(* CODESYS project T620X_PLC_CR711S.project
   Title: T620X PLC
   Description: T620X PLC - pwm ramp mods / sim mods - link fixed for RAMP_LIMIT to the output block
   Version: 1.0.3.0
   Company: Mtech

Project tree, tasks and I/O mapping:
  SafetyPLC : CR711S SIL2, ifm electronic, order no. CR711S, version 3.2.0.0
    application Application
      libraries: ifmR360-3, * (ifm electronic); Standard, * (System); Util, * (System)
      task Task (cyclic, interval t#10ms, priority 1, watchdog t#8ms x 1) calls PLC_PRG
      global variables EVL
      program PLC_PRG [FBD]
    Communication : Communication, ifm electronic, version 3.2.0.0
      CAN : CAN, ifm electronic, version 3.2.0.0
      Ethernet : Ethernet, ifm electronic, version 3.2.0.0
    HMI : HMI, ifm electronic, version 3.2.0.0
      User_LEDs : User_LEDs, ifm electronic, version 3.2.0.0
          input  UserLED0_I : LED_IEC_B_INPUT_MAPPING_TYPE  // UserLED0_I
          input  UserLED1_I : LED_IEC_B_INPUT_MAPPING_TYPE  // UserLED1_I
          input  UserLED2_I : LED_IEC_B_INPUT_MAPPING_TYPE  // UserLED2_I
          input  UserLED3_I : LED_IEC_B_INPUT_MAPPING_TYPE  // UserLED3_I
          output UserLED0_Q : LED_IEC_B_OUTPUT_MAPPING_TYPE  // User LED 0
          output UserLED1_Q : LED_IEC_B_OUTPUT_MAPPING_TYPE  // User LED 1
          output UserLED2_Q : LED_IEC_B_OUTPUT_MAPPING_TYPE  // User LED 2
          output UserLED3_Q : LED_IEC_B_OUTPUT_MAPPING_TYPE  // User LED 3
    Local_IO : Local_IO, ifm electronic, version 3.2.0.0
      Inputs : Inputs, ifm electronic, version 3.2.0.0
          input  IN0100_I : IN_MULTIFUNCTION_A_INPUT_MAPPING_TYPE  // IN0100_I
          input  IN0101_I : IN_MULTIFUNCTION_A_INPUT_MAPPING_TYPE  // IN0101_I
          input  IN0102_I : IN_MULTIFUNCTION_A_INPUT_MAPPING_TYPE  // IN0102_I
          input  IN0103_I : IN_MULTIFUNCTION_A_INPUT_MAPPING_TYPE  // IN0103_I
          input  IN0200_I : IN_MULTIFUNCTION_A_INPUT_MAPPING_TYPE  // IN0200_I
          input  IN0201_I : IN_MULTIFUNCTION_A_INPUT_MAPPING_TYPE  // IN0201_I
          input  IN0202_I : IN_MULTIFUNCTION_A_INPUT_MAPPING_TYPE  // IN0202_I
          input  IN0203_I : IN_MULTIFUNCTION_A_INPUT_MAPPING_TYPE  // IN0203_I
          input  IN0600_I : IN_MULTIFUNCTION_A_INPUT_MAPPING_TYPE  // IN0600_I
          input  IN0601_I : IN_MULTIFUNCTION_A_INPUT_MAPPING_TYPE  // IN0601_I
          input  IN0602_I : IN_MULTIFUNCTION_A_INPUT_MAPPING_TYPE  // IN0602_I
          input  IN0603_I : IN_MULTIFUNCTION_A_INPUT_MAPPING_TYPE  // IN0603_I
          input  IN0700_I : IN_MULTIFUNCTION_A_INPUT_MAPPING_TYPE  // IN0700_I
          input  IN0701_I : IN_MULTIFUNCTION_A_INPUT_MAPPING_TYPE  // IN0701_I
          input  IN0702_I : IN_MULTIFUNCTION_A_INPUT_MAPPING_TYPE  // IN0702_I
          input  IN0703_I : IN_MULTIFUNCTION_A_INPUT_MAPPING_TYPE  // IN0703_I
          input  IN0400_I : IN_RESISTOR_A_INPUT_MAPPING_TYPE  // IN0400_I
          input  IN0401_I : IN_RESISTOR_A_INPUT_MAPPING_TYPE  // IN0401_I
          input  IN0900_I : IN_RESISTOR_A_INPUT_MAPPING_TYPE  // IN0900_I
          input  IN0901_I : IN_RESISTOR_A_INPUT_MAPPING_TYPE  // IN0901_I
          input  IN0300_I : IN_DIGITAL_B_INPUT_MAPPING_TYPE  // IN0300_I
          input  IN0301_I : IN_DIGITAL_B_INPUT_MAPPING_TYPE  // IN0301_I
          input  IN0800_I : IN_DIGITAL_B_INPUT_MAPPING_TYPE  // IN0800_I
          input  IN0801_I : IN_DIGITAL_B_INPUT_MAPPING_TYPE  // IN0801_I
          input  COM_RESET_I : IN_COMMUNICATION_RESET_INPUT_MAPPING_TYPE  // COM_RESET_I
          input  IN0000_I : IN_FREQUENCY_B_CHANNEL_A_INPUT_MAPPING_TYPE  // IN0000_I
          input  IN0002_I : IN_FREQUENCY_B_CHANNEL_A_INPUT_MAPPING_TYPE  // IN0002_I
          input  IN0500_I : IN_FREQUENCY_B_CHANNEL_A_INPUT_MAPPING_TYPE  // IN0500_I
          input  IN0502_I : IN_FREQUENCY_B_CHANNEL_A_INPUT_MAPPING_TYPE  // IN0502_I
          input  IN0001_I : IN_FREQUENCY_B_CHANNEL_B_INPUT_MAPPING_TYPE  // IN0001_I
          input  IN0003_I : IN_FREQUENCY_B_CHANNEL_B_INPUT_MAPPING_TYPE  // IN0003_I
          input  IN0501_I : IN_FREQUENCY_B_CHANNEL_B_INPUT_MAPPING_TYPE  // IN0501_I
          input  IN0503_I : IN_FREQUENCY_B_CHANNEL_B_INPUT_MAPPING_TYPE  // IN0503_I
      Outputs : Outputs, ifm electronic, version 3.2.0.0
          input  OUT0006_I : OUT_PWM_40_BRIDGE_A_INPUT_MAPPING_TYPE  // OUT0006_I
          input  OUT0106_I : OUT_PWM_40_BRIDGE_A_INPUT_MAPPING_TYPE  // OUT0106_I
          input  OUT0206_I : OUT_PWM_40_BRIDGE_A_INPUT_MAPPING_TYPE  // OUT0206_I
          input  OUT0008_I : OUT_PWM_40_A_INPUT_MAPPING_TYPE  // OUT0008_I
          input  OUT0108_I : OUT_PWM_40_A_INPUT_MAPPING_TYPE  // OUT0108_I
          input  OUT0208_I : OUT_PWM_40_A_INPUT_MAPPING_TYPE  // OUT0208_I
          input  OUT0000_I : OUT_PWM_25_A_INPUT_MAPPING_TYPE  // OUT0000_I
          input  OUT0002_I : OUT_PWM_25_A_INPUT_MAPPING_TYPE  // OUT0002_I
          input  OUT0004_I : OUT_PWM_25_A_INPUT_MAPPING_TYPE  // OUT0004_I
          input  OUT0100_I : OUT_PWM_25_A_INPUT_MAPPING_TYPE  // OUT0100_I
          input  OUT0102_I : OUT_PWM_25_A_INPUT_MAPPING_TYPE  // OUT0102_I
          input  OUT0104_I : OUT_PWM_25_A_INPUT_MAPPING_TYPE  // OUT0104_I
          input  OUT0200_I : OUT_PWM_25_A_INPUT_MAPPING_TYPE  // OUT0200_I
          input  OUT0202_I : OUT_PWM_25_A_INPUT_MAPPING_TYPE  // OUT0202_I
          input  OUT0204_I : OUT_PWM_25_A_INPUT_MAPPING_TYPE  // OUT0204_I
          input  OUT3001_I : OUT_VOLTAGE_A_INPUT_MAPPING_TYPE  // OUT3001_I
          input  OUT3000_I : OUT_SUPPLY_A_INPUT_MAPPING_TYPE  // OUT3000_I
          input  OUT0001_I : OUT_PWM_25_B_INPUT_MAPPING_TYPE  // OUT0001_I
          input  OUT0003_I : OUT_PWM_25_B_INPUT_MAPPING_TYPE  // OUT0003_I
          input  OUT0005_I : OUT_PWM_25_B_INPUT_MAPPING_TYPE  // OUT0005_I
          input  OUT0101_I : OUT_PWM_25_B_INPUT_MAPPING_TYPE  // OUT0101_I
          input  OUT0103_I : OUT_PWM_25_B_INPUT_MAPPING_TYPE  // OUT0103_I
          input  OUT0105_I : OUT_PWM_25_B_INPUT_MAPPING_TYPE  // OUT0105_I
          input  OUT0201_I : OUT_PWM_25_B_INPUT_MAPPING_TYPE  // OUT0201_I
          input  OUT0203_I : OUT_PWM_25_B_INPUT_MAPPING_TYPE  // OUT0203_I
          input  OUT0205_I : OUT_PWM_25_B_INPUT_MAPPING_TYPE  // OUT0205_I
          input  OUT0007_I : OUT_PWM_40_BRIDGE_A_INPUT_MAPPING_TYPE  // OUT0007_I
          input  OUT0107_I : OUT_PWM_40_BRIDGE_A_INPUT_MAPPING_TYPE  // OUT0107_I
          input  OUT0207_I : OUT_PWM_40_BRIDGE_A_INPUT_MAPPING_TYPE  // OUT0207_I
          output OUT0006_Q : OUT_PWM_40_BRIDGE_A_OUTPUT_MAPPING_TYPE  // OUT0006_Q
          output OUT0106_Q : OUT_PWM_40_BRIDGE_A_OUTPUT_MAPPING_TYPE  // OUT0106_Q
          output OUT0206_Q : OUT_PWM_40_BRIDGE_A_OUTPUT_MAPPING_TYPE  // OUT0206_Q
          output OUT0008_Q : OUT_PWM_40_A_OUTPUT_MAPPING_TYPE  // OUT0008_Q
          output OUT0108_Q : OUT_PWM_40_A_OUTPUT_MAPPING_TYPE  // OUT0108_Q
          output OUT0208_Q : OUT_PWM_40_A_OUTPUT_MAPPING_TYPE  // OUT0208_Q
          output OUT0000_Q : OUT_PWM_25_A_OUTPUT_MAPPING_TYPE  // OUT0000_Q
          output OUT0002_Q : OUT_PWM_25_A_OUTPUT_MAPPING_TYPE  // OUT0002_Q
          output OUT0004_Q : OUT_PWM_25_A_OUTPUT_MAPPING_TYPE  // OUT0004_Q
          output OUT0100_Q : OUT_PWM_25_A_OUTPUT_MAPPING_TYPE  // OUT0100_Q
          output OUT0102_Q : OUT_PWM_25_A_OUTPUT_MAPPING_TYPE  // OUT0102_Q
          output OUT0104_Q : OUT_PWM_25_A_OUTPUT_MAPPING_TYPE  // OUT0104_Q
          output OUT0200_Q : OUT_PWM_25_A_OUTPUT_MAPPING_TYPE  // OUT0200_Q
          output OUT0202_Q : OUT_PWM_25_A_OUTPUT_MAPPING_TYPE  // OUT0202_Q
          output OUT0204_Q : OUT_PWM_25_A_OUTPUT_MAPPING_TYPE  // OUT0204_Q
          output OUT3001_Q : OUT_VOLTAGE_A_OUTPUT_MAPPING_TYPE  // OUT3001_Q
          output OUT3000_Q : OUT_SUPPLY_A_OUTPUT_MAPPING_TYPE  // OUT3000_Q
          output OUT0001_Q : OUT_PWM_25_B_OUTPUT_MAPPING_TYPE  // OUT0001_Q
          output OUT0003_Q : OUT_PWM_25_B_OUTPUT_MAPPING_TYPE  // OUT0003_Q
          output OUT0005_Q : OUT_PWM_25_B_OUTPUT_MAPPING_TYPE  // OUT0005_Q
          output OUT0101_Q : OUT_PWM_25_B_OUTPUT_MAPPING_TYPE  // OUT0101_Q
          output OUT0103_Q : OUT_PWM_25_B_OUTPUT_MAPPING_TYPE  // OUT0103_Q
          output OUT0105_Q : OUT_PWM_25_B_OUTPUT_MAPPING_TYPE  // OUT0105_Q
          output OUT0201_Q : OUT_PWM_25_B_OUTPUT_MAPPING_TYPE  // OUT0201_Q
          output OUT0203_Q : OUT_PWM_25_B_OUTPUT_MAPPING_TYPE  // OUT0203_Q
          output OUT0205_Q : OUT_PWM_25_B_OUTPUT_MAPPING_TYPE  // OUT0205_Q
          output OUT0007_Q : OUT_PWM_40_BRIDGE_A_OUTPUT_MAPPING_TYPE  // OUT0007_Q
          output OUT0107_Q : OUT_PWM_40_BRIDGE_A_OUTPUT_MAPPING_TYPE  // OUT0107_Q
          output OUT0207_Q : OUT_PWM_40_BRIDGE_A_OUTPUT_MAPPING_TYPE  // OUT0207_Q
      System_Inputs : System_Inputs, ifm electronic, version 3.2.0.0
          input  VBB30 : IN_SYSTEM_VOLTAGE_INPUT_MAPPING_TYPE  // VBB30
          input  VBB15 : IN_SYSTEM_VOLTAGE_INPUT_MAPPING_TYPE  // VBB15
          input  TemperatureBoard0 : IN_TEMPERATURE_INPUT_MAPPING_TYPE  // TemperatureBoard0
          input  TemperatureChip0 : IN_TEMPERATURE_INPUT_MAPPING_TYPE  // TemperatureChip0
      System_Outputs : System_Outputs, ifm electronic, version 3.2.0.0
          input  VBB0_SW_I : OUT_GROUP_SWITCH_INPUT_MAPPING_TYPE  // VBB0_SW_I
          input  VBB1_SW_I : OUT_GROUP_SWITCH_INPUT_MAPPING_TYPE  // VBB1_SW_I
          input  VBB2_SW_I : OUT_GROUP_SWITCH_INPUT_MAPPING_TYPE  // VBB2_SW_I
          output VBB0_SW_Q : OUT_GROUP_SWITCH_OUTPUT_MAPPING_TYPE  // VBB0_SW_Q
          output VBB1_SW_Q : OUT_GROUP_SWITCH_OUTPUT_MAPPING_TYPE  // VBB1_SW_Q
          output VBB2_SW_Q : OUT_GROUP_SWITCH_OUTPUT_MAPPING_TYPE  // VBB2_SW_Q
          output SUPPLY_SWITCH_Q : OUT_SYS_SWITCH_OUTPUT_MAPPING_TYPE  // SUPPLY_SWITCH_Q
  StandardPLC : CR711S Standard, ifm electronic, order no. CR711S, version 3.2.0.0
    application Application
      libraries: ifmR360-3, * (ifm electronic); Standard, * (System); Util, * (System); PIL Master Library, 1.0.0 (Powerhouse IRL Ltd); SLL_IFM_Version, 0.0.0.2 (SLL)
      task Task (cyclic, interval t#10ms, priority 1, watchdog t#8ms x 1) calls PLC_PRG
      EVC
      program PLC_PRG [FBD]
      program config_IO [FBD]
      global variables GVL
      program EngineRun [FBD]
      CAN Comms/
        Engine Comms/
          function block CounterChecksum [ST]
          function block DM1_Condition [FBD]
          program Engine_Coms [FBD]
          function block fb_Extract_SPN [FBD]
          function block Pack2bits [ST]
        program CAN_COMS [FBD]
      program Alarms [FBD]
      program FanCtrl [FBD]
      global variables RetVal
      Control/
        program Tracking [FBD]
        program Auto_Sequence [FBD]
        program ManualSequence [FBD]
        program JackLegs [FBD]
      function block fbSmoothing [ST]
      Set Points/
        function block SP_CountX1 [FBD]
        program SetPoints [FBD]
        function block SP_CountX10 [FBD]
      global variables SIM
      program SIM_MAIN [FBD]
      program PLC_Version [FBD]
    Communication : Communication, ifm electronic, version 3.2.0.0
      CAN : CAN, ifm electronic, version 3.2.0.0
      Ethernet : Ethernet, ifm electronic, version 3.2.0.0
    HMI : HMI, ifm electronic, version 3.2.0.0
      User_LEDs : User_LEDs, ifm electronic, version 3.2.0.0
          input  UserLED0_I : LED_IEC_B_INPUT_MAPPING_TYPE  // UserLED0_I
          input  UserLED1_I : LED_IEC_B_INPUT_MAPPING_TYPE  // UserLED1_I
          input  UserLED2_I : LED_IEC_B_INPUT_MAPPING_TYPE  // UserLED2_I
          input  UserLED3_I : LED_IEC_B_INPUT_MAPPING_TYPE  // UserLED3_I
          output UserLED0_Q : LED_IEC_B_OUTPUT_MAPPING_TYPE  // User LED 0
          output UserLED1_Q : LED_IEC_B_OUTPUT_MAPPING_TYPE  // User LED 1
          output UserLED2_Q : LED_IEC_B_OUTPUT_MAPPING_TYPE  // User LED 2
          output UserLED3_Q : LED_IEC_B_OUTPUT_MAPPING_TYPE  // User LED 3
    Local_IO : Local_IO, ifm electronic, version 3.2.0.0
      Inputs : Inputs, ifm electronic, version 3.2.0.0
          input  IN0100_I : IN_MULTIFUNCTION_A_INPUT_MAPPING_TYPE  // IN0100_I
          input  IN0101_I : IN_MULTIFUNCTION_A_INPUT_MAPPING_TYPE  // IN0101_I
          input  IN0102_I : IN_MULTIFUNCTION_A_INPUT_MAPPING_TYPE  // IN0102_I
          input  IN0103_I : IN_MULTIFUNCTION_A_INPUT_MAPPING_TYPE  // IN0103_I
          input  IN0200_I : IN_MULTIFUNCTION_A_INPUT_MAPPING_TYPE  // IN0200_I
          input  IN0201_I : IN_MULTIFUNCTION_A_INPUT_MAPPING_TYPE  // IN0201_I
          input  IN0202_I : IN_MULTIFUNCTION_A_INPUT_MAPPING_TYPE  // IN0202_I
          input  IN0203_I : IN_MULTIFUNCTION_A_INPUT_MAPPING_TYPE  // IN0203_I
          input  IN0600_I : IN_MULTIFUNCTION_A_INPUT_MAPPING_TYPE  // IN0600_I
          input  IN0601_I : IN_MULTIFUNCTION_A_INPUT_MAPPING_TYPE  // IN0601_I
          input  IN0602_I : IN_MULTIFUNCTION_A_INPUT_MAPPING_TYPE  // IN0602_I
          input  IN0603_I : IN_MULTIFUNCTION_A_INPUT_MAPPING_TYPE  // IN0603_I
          input  IN0700_I : IN_MULTIFUNCTION_A_INPUT_MAPPING_TYPE  // IN0700_I
          input  IN0701_I : IN_MULTIFUNCTION_A_INPUT_MAPPING_TYPE  // IN0701_I
          input  IN0702_I : IN_MULTIFUNCTION_A_INPUT_MAPPING_TYPE  // IN0702_I
          input  IN0703_I : IN_MULTIFUNCTION_A_INPUT_MAPPING_TYPE  // IN0703_I
          input  IN0400_I : IN_RESISTOR_A_INPUT_MAPPING_TYPE  // IN0400_I
          input  IN0401_I : IN_RESISTOR_A_INPUT_MAPPING_TYPE  // IN0401_I
          input  IN0900_I : IN_RESISTOR_A_INPUT_MAPPING_TYPE  // IN0900_I
          input  IN0901_I : IN_RESISTOR_A_INPUT_MAPPING_TYPE  // IN0901_I
          input  IN0300_I : IN_DIGITAL_B_INPUT_MAPPING_TYPE  // IN0300_I
          input  IN0301_I : IN_DIGITAL_B_INPUT_MAPPING_TYPE  // IN0301_I
          input  IN0800_I : IN_DIGITAL_B_INPUT_MAPPING_TYPE  // IN0800_I
          input  IN0801_I : IN_DIGITAL_B_INPUT_MAPPING_TYPE  // IN0801_I
          input  COM_RESET_I : IN_COMMUNICATION_RESET_INPUT_MAPPING_TYPE  // COM_RESET_I
          input  IN0000_I : IN_FREQUENCY_B_CHANNEL_A_INPUT_MAPPING_TYPE  // IN0000_I
          input  IN0002_I : IN_FREQUENCY_B_CHANNEL_A_INPUT_MAPPING_TYPE  // IN0002_I
          input  IN0500_I : IN_FREQUENCY_B_CHANNEL_A_INPUT_MAPPING_TYPE  // IN0500_I
          input  IN0502_I : IN_FREQUENCY_B_CHANNEL_A_INPUT_MAPPING_TYPE  // IN0502_I
          input  IN0001_I : IN_FREQUENCY_B_CHANNEL_B_INPUT_MAPPING_TYPE  // IN0001_I
          input  IN0003_I : IN_FREQUENCY_B_CHANNEL_B_INPUT_MAPPING_TYPE  // IN0003_I
          input  IN0501_I : IN_FREQUENCY_B_CHANNEL_B_INPUT_MAPPING_TYPE  // IN0501_I
          input  IN0503_I : IN_FREQUENCY_B_CHANNEL_B_INPUT_MAPPING_TYPE  // IN0503_I
      Outputs : Outputs, ifm electronic, version 3.2.0.0
          input  OUT0006_I : OUT_PWM_40_BRIDGE_A_INPUT_MAPPING_TYPE  // OUT0006_I
          input  OUT0106_I : OUT_PWM_40_BRIDGE_A_INPUT_MAPPING_TYPE  // OUT0106_I
          input  OUT0206_I : OUT_PWM_40_BRIDGE_A_INPUT_MAPPING_TYPE  // OUT0206_I
          input  OUT0008_I : OUT_PWM_40_A_INPUT_MAPPING_TYPE  // OUT0008_I
          input  OUT0108_I : OUT_PWM_40_A_INPUT_MAPPING_TYPE  // OUT0108_I
          input  OUT0208_I : OUT_PWM_40_A_INPUT_MAPPING_TYPE  // OUT0208_I
          input  OUT0000_I : OUT_PWM_25_A_INPUT_MAPPING_TYPE  // OUT0000_I
          input  OUT0002_I : OUT_PWM_25_A_INPUT_MAPPING_TYPE  // OUT0002_I
          input  OUT0004_I : OUT_PWM_25_A_INPUT_MAPPING_TYPE  // OUT0004_I
          input  OUT0100_I : OUT_PWM_25_A_INPUT_MAPPING_TYPE  // OUT0100_I
          input  OUT0102_I : OUT_PWM_25_A_INPUT_MAPPING_TYPE  // OUT0102_I
          input  OUT0104_I : OUT_PWM_25_A_INPUT_MAPPING_TYPE  // OUT0104_I
          input  OUT0200_I : OUT_PWM_25_A_INPUT_MAPPING_TYPE  // OUT0200_I
          input  OUT0202_I : OUT_PWM_25_A_INPUT_MAPPING_TYPE  // OUT0202_I
          input  OUT0204_I : OUT_PWM_25_A_INPUT_MAPPING_TYPE  // OUT0204_I
          input  OUT3001_I : OUT_VOLTAGE_A_INPUT_MAPPING_TYPE  // OUT3001_I
          input  OUT3000_I : OUT_SUPPLY_A_INPUT_MAPPING_TYPE  // OUT3000_I
          input  OUT0001_I : OUT_PWM_25_B_INPUT_MAPPING_TYPE  // OUT0001_I
          input  OUT0003_I : OUT_PWM_25_B_INPUT_MAPPING_TYPE  // OUT0003_I
          input  OUT0005_I : OUT_PWM_25_B_INPUT_MAPPING_TYPE  // OUT0005_I
          input  OUT0101_I : OUT_PWM_25_B_INPUT_MAPPING_TYPE  // OUT0101_I
          input  OUT0103_I : OUT_PWM_25_B_INPUT_MAPPING_TYPE  // OUT0103_I
          input  OUT0105_I : OUT_PWM_25_B_INPUT_MAPPING_TYPE  // OUT0105_I
          input  OUT0201_I : OUT_PWM_25_B_INPUT_MAPPING_TYPE  // OUT0201_I
          input  OUT0203_I : OUT_PWM_25_B_INPUT_MAPPING_TYPE  // OUT0203_I
          input  OUT0205_I : OUT_PWM_25_B_INPUT_MAPPING_TYPE  // OUT0205_I
          input  OUT0007_I : OUT_PWM_40_BRIDGE_A_INPUT_MAPPING_TYPE  // OUT0007_I
          input  OUT0107_I : OUT_PWM_40_BRIDGE_A_INPUT_MAPPING_TYPE  // OUT0107_I
          input  OUT0207_I : OUT_PWM_40_BRIDGE_A_INPUT_MAPPING_TYPE  // OUT0207_I
          output OUT0006_Q : OUT_PWM_40_BRIDGE_A_OUTPUT_MAPPING_TYPE  // OUT0006_Q
          output OUT0106_Q : OUT_PWM_40_BRIDGE_A_OUTPUT_MAPPING_TYPE  // OUT0106_Q
          output OUT0206_Q : OUT_PWM_40_BRIDGE_A_OUTPUT_MAPPING_TYPE  // OUT0206_Q
          output OUT0008_Q : OUT_PWM_40_A_OUTPUT_MAPPING_TYPE  // OUT0008_Q
          output OUT0108_Q : OUT_PWM_40_A_OUTPUT_MAPPING_TYPE  // OUT0108_Q
          output OUT0208_Q : OUT_PWM_40_A_OUTPUT_MAPPING_TYPE  // OUT0208_Q
          output OUT0000_Q : OUT_PWM_25_A_OUTPUT_MAPPING_TYPE  // OUT0000_Q
          output OUT0002_Q : OUT_PWM_25_A_OUTPUT_MAPPING_TYPE  // OUT0002_Q
          output OUT0004_Q : OUT_PWM_25_A_OUTPUT_MAPPING_TYPE  // OUT0004_Q
          output OUT0100_Q : OUT_PWM_25_A_OUTPUT_MAPPING_TYPE  // OUT0100_Q
          output OUT0102_Q : OUT_PWM_25_A_OUTPUT_MAPPING_TYPE  // OUT0102_Q
          output OUT0104_Q : OUT_PWM_25_A_OUTPUT_MAPPING_TYPE  // OUT0104_Q
          output OUT0200_Q : OUT_PWM_25_A_OUTPUT_MAPPING_TYPE  // OUT0200_Q
          output OUT0202_Q : OUT_PWM_25_A_OUTPUT_MAPPING_TYPE  // OUT0202_Q
          output OUT0204_Q : OUT_PWM_25_A_OUTPUT_MAPPING_TYPE  // OUT0204_Q
          output OUT3001_Q : OUT_VOLTAGE_A_OUTPUT_MAPPING_TYPE  // OUT3001_Q
          output OUT3000_Q : OUT_SUPPLY_A_OUTPUT_MAPPING_TYPE  // OUT3000_Q
          output OUT0001_Q : OUT_PWM_25_B_OUTPUT_MAPPING_TYPE  // OUT0001_Q
          output OUT0003_Q : OUT_PWM_25_B_OUTPUT_MAPPING_TYPE  // OUT0003_Q
          output OUT0005_Q : OUT_PWM_25_B_OUTPUT_MAPPING_TYPE  // OUT0005_Q
          output OUT0101_Q : OUT_PWM_25_B_OUTPUT_MAPPING_TYPE  // OUT0101_Q
          output OUT0103_Q : OUT_PWM_25_B_OUTPUT_MAPPING_TYPE  // OUT0103_Q
          output OUT0105_Q : OUT_PWM_25_B_OUTPUT_MAPPING_TYPE  // OUT0105_Q
          output OUT0201_Q : OUT_PWM_25_B_OUTPUT_MAPPING_TYPE  // OUT0201_Q
          output OUT0203_Q : OUT_PWM_25_B_OUTPUT_MAPPING_TYPE  // OUT0203_Q
          output OUT0205_Q : OUT_PWM_25_B_OUTPUT_MAPPING_TYPE  // OUT0205_Q
          output OUT0007_Q : OUT_PWM_40_BRIDGE_A_OUTPUT_MAPPING_TYPE  // OUT0007_Q
          output OUT0107_Q : OUT_PWM_40_BRIDGE_A_OUTPUT_MAPPING_TYPE  // OUT0107_Q
          output OUT0207_Q : OUT_PWM_40_BRIDGE_A_OUTPUT_MAPPING_TYPE  // OUT0207_Q
      System_Inputs : System_Inputs, ifm electronic, version 3.2.0.0
          input  VBB30 AT %IW251 : IN_SYSTEM_VOLTAGE_INPUT_MAPPING_TYPE  // VBB30
          input  VBB15 : IN_SYSTEM_VOLTAGE_INPUT_MAPPING_TYPE  // VBB15
          input  TemperatureBoard0 : IN_TEMPERATURE_INPUT_MAPPING_TYPE  // TemperatureBoard0
          input  TemperatureChip0 : IN_TEMPERATURE_INPUT_MAPPING_TYPE  // TemperatureChip0
      System_Outputs : System_Outputs, ifm electronic, version 3.2.0.0
          input  VBB0_SW_I : OUT_GROUP_SWITCH_INPUT_MAPPING_TYPE  // VBB0_SW_I
          input  VBB1_SW_I : OUT_GROUP_SWITCH_INPUT_MAPPING_TYPE  // VBB1_SW_I
          input  VBB2_SW_I : OUT_GROUP_SWITCH_INPUT_MAPPING_TYPE  // VBB2_SW_I
          output VBB0_SW_Q : OUT_GROUP_SWITCH_OUTPUT_MAPPING_TYPE  // VBB0_SW_Q
          output VBB1_SW_Q : OUT_GROUP_SWITCH_OUTPUT_MAPPING_TYPE  // VBB1_SW_Q
          output VBB2_SW_Q : OUT_GROUP_SWITCH_OUTPUT_MAPPING_TYPE  // VBB2_SW_Q
          output SUPPLY_SWITCH_Q : OUT_SYS_SWITCH_OUTPUT_MAPPING_TYPE  // SUPPLY_SWITCH_Q
  CR711S : CR711S, ifm electronic, order no. CR711S, version 3.2.0.0
  Project Information/
    function GetCompany [ST]
    function GetTitle [ST]
    function GetVersion [ST]
    function GetTextProperty [ST]
    function GetTextProperty2 [ST]
    function GetNumberProperty [ST]
    function GetBooleanProperty [ST]
    function GetVersionProperty [ST]
*)

// SafetyPLC/Application/EVL
(* THIS EVL IS AUTOGENERATED. DO NOT MODIFY THESE ATTRIBUTES. *)
{attribute 'location' := '16#800' }
{attribute 'linkalways'}
{attribute 'qualified_only'}
VAR_GLOBAL

END_VAR

// StandardPLC/Application/GVL
{attribute 'qualified_only'}
VAR_GLOBAL
	HalfSecBlink: BOOL;
	OneSecBlink: BOOL;
	KEY_F1: BOOL;
	KEY_F2: BOOL;
	KEY_F3: BOOL;
	KEY_F4: BOOL;
	KEY_F5: BOOL;
	KEY_F6: BOOL;
	KEY_UP: BOOL;
	KEY_DOWN: BOOL;
	KEY_LEFT: BOOL;
	KEY_RIGHT: BOOL;
	KEY_OK: BOOL;
	RT_F1: BOOL;
	RT_F2: BOOL;
	RT_F3: BOOL;
	RT_F4: BOOL;
	RT_F5: BOOL;
	RT_F6: BOOL;
	RT_UP: BOOL;
	RT_DOWN: BOOL;
	RT_LEFT: BOOL;
	RT_RIGHT: BOOL;
	RT_OK: BOOL;
	Page1Selected: BOOL;
	Page2Selected: BOOL;
	Page3Selected: BOOL;
	Page4Selected: BOOL;
	Page5Selected: BOOL;
	Page6Selected: BOOL;
	Page10Selected: BOOL;
	Page11Selected: BOOL;
	Page12Selected: BOOL;
	
	Reset: BOOL;
	EStop_OK: BOOL;
	ThermoStat: BOOL;
	RHS_TrommelDoorSw: BOOL;
	LHS_TrommelDoorSw: BOOL;
	HydOilTemp_Sw: BOOL;
	HydOilLevel_Sw: BOOL;
	RadioRHS_JackLegRaise_Req: BOOL;
	RadioRHS_JackLegLower_Req: BOOL;
	RadioLHS_JackLegRaise_Req: BOOL;
	RadioLHS_JackLegLower_Req: BOOL;
	RadioSideConvRaiseReq: BOOL;
	RadioSideConvLowerReq: BOOL;
	UmbTrackReq: BOOL;
	UmbMachineStop: BOOL;
	RTF_Req: BOOL;
	RTR_Req: BOOL;
	LTF_Req: BOOL;
	LTR_Req: BOOL;
	TailConvSpd_mA: UINT;
	TailConvOn_OP: BOOL;
	SideConvSpd_mA: UINT;
	SideConvOn_OP: BOOL;
	SideTransferSpd_mA: UINT;
	SideTransferOn_OP: BOOL;
	SetupDumpValve_OP: BOOL;
	CollectionConvSpd_mA: UINT;
	CollectionConvOn_OP: BOOL;
	DrumSpd_mA: UINT;
	DrumSpd_mA_RAMP_LIMIT: UINT;
	DrumOnOff_OP: BOOL;
	FeederSpd_mA: UINT;
	FeederOnOff_OP: BOOL;
	DivertOilToTrack_OP: BOOL;
	RHS_JackLegRaise_OP: BOOL;
	RHS_JackLegLower_OP: BOOL;
	LHS_JackLegRaise_OP: BOOL;
	LHS_JackLegLower_OP: BOOL;
	LeftTrackDivert_OP: BOOL;
	LTF_OP: BOOL;
	LTR_OP: BOOL;
	RightTrackDivert_OP: BOOL;
	RTF_OP: BOOL;
	RTR_OP: BOOL;
	EngineRunning: BOOL;
	ECUenable: BOOL;
	CrankEnable: BOOL;
	RequestedRPM: WORD;
	TrackingMode: BOOL;
	CriticalShutdown: BOOL;
	DefLowLevLamp: BOOL;
	VBB30_mV: WORD;
	VBB0_mV: WORD;
	VBB1_mV: WORD;
	VBB2_mV: WORD;
	ChargeLamp: BOOL;
	UmbMachineShutdown: BOOL;
	LowOilPressAlarm: BOOL;
	EngineHiTempAlarm: BOOL;
	LowHydOilAlarm: BOOL;
	HydTempAlarm: BOOL;
	FanFwd_OP: BOOL;
	FanRev_OP: BOOL;
	SideConvRaise_OP: BOOL;
	SideConvLower_OP: BOOL;
	AutoStopMode: BOOL;
	AutoMode: BOOL;
	DisplayAutoStop: BOOL;
	AutoShutdownAlarm: BOOL;
	DisplayAutoStarting: BOOL;
	SetupMode: BOOL;
	ReqJackLegs: BOOL;
	ReqHydSetup: BOOL;
	ManualMode: BOOL;
	FuelLevel_Percent: BYTE;
	LowFuelWarn: BOOL;
	LowFuelAlarm: BOOL;
	DrumPress_bar: REAL;
	DrumHighPress_Warn: BOOL;
	DrumHighPress_Alarm: BOOL;
END_VAR

// StandardPLC/Application/RetVal
{attribute 'qualified_only'}
VAR_GLOBAL PERSISTENT RETAIN
	FwdTime_sec: WORD;
	RevTime_sec: WORD;
	TailConvSpd_Percent: BYTE:=100;
	SideConvSpd_Percent: BYTE:=100;
	SideTransferConvSpd_Percent: BYTE:=100;
	CollectConvSpd_Percent: BYTE:=100;
	DrumSpd_Percent: BYTE:=100;
	FeederSpd_Percent: BYTE:=100;
	TailConvSpd_Min_mA: INT:=500;
	TailConvSpd_Max_mA: INT:=1450;
	SideConvSpd_Min_mA: INT:=500;
	SideConvSpd_Max_mA: INT:=1450;
	SideTransferConvSpd_Min_mA: INT:=500;
	SideTransferConvSpd_Max_mA: INT:=1450;
	CollectConvSpd_Min_mA: INT:=500;
	CollectConvSpd_Max_mA: INT:=1450;
	DrumSpd_Min_mA: INT:=500;
	DrumSpd_Max_mA: INT:=1450;
	FeederSpd_Min_mA: INT:=500;
	FeederSpd_Max_mA: INT:=1450;
	EnableDrumPressCutOut: BOOL:=TRUE;
	DrumPressReset_SP_bar: BYTE:=150;
	DrumPressHi_SP_bar: BYTE:=160;
	DrumPressHiHi_SP_bar: BYTE:=165;
END_VAR

// StandardPLC/Application/SIM
{attribute 'qualified_only'}
VAR_GLOBAL
	SIM_SETUP: BOOL;
	
	SIM_SKIP_IO_CONFIG: BOOL;
	
	ESTOP_VALUE: BOOL:=TRUE;
	
	ADBLUE_ENA:BOOL;
	ADBLUE_VALUE:BYTE:=30;
	
	ENGINE_ENA: BOOL;
	ENGINE_VALUE : WORD:=800;	
END_VAR

// SafetyPLC/Application/PLC_PRG
PROGRAM PLC_PRG
VAR
END_VAR

// NETWORK 1

END_PROGRAM

// StandardPLC/Application/PLC_PRG
PROGRAM PLC_PRG
VAR
	init: BOOL := TRUE;
	Blink_0: Blink;
	Blink_1: Blink;
END_VAR

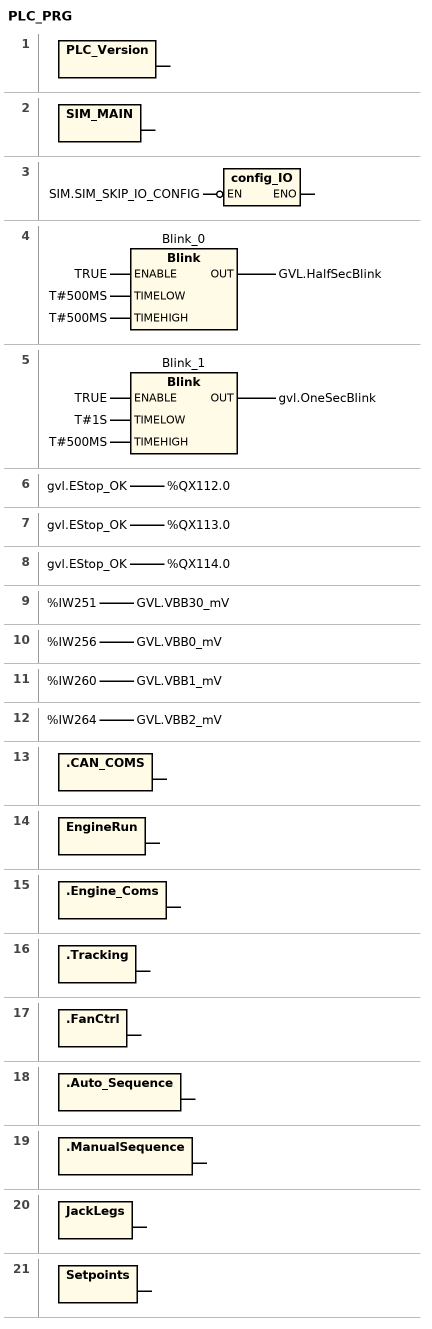
// NETWORK 1
PLC_Version();

// NETWORK 2
SIM_MAIN();

// NETWORK 3
IF NOT SIM.SIM_SKIP_IO_CONFIG THEN config_IO(); END_IF

// NETWORK 4
Blink_0(ENABLE := TRUE, TIMELOW := T#500MS, TIMEHIGH := T#500MS); // Blink
GVL.HalfSecBlink := Blink_0.OUT;

// NETWORK 5
Blink_1(ENABLE := TRUE, TIMELOW := T#1S, TIMEHIGH := T#500MS); // Blink
gvl.OneSecBlink := Blink_1.OUT;

// NETWORK 6
%QX112.0 := gvl.EStop_OK;

// NETWORK 7
%QX113.0 := gvl.EStop_OK;

// NETWORK 8
%QX114.0 := gvl.EStop_OK;

// NETWORK 9
GVL.VBB30_mV := %IW251;

// NETWORK 10
GVL.VBB0_mV := %IW256;

// NETWORK 11
GVL.VBB1_mV := %IW260;

// NETWORK 12
GVL.VBB2_mV := %IW264;

// NETWORK 13
.CAN_COMS();

// NETWORK 14
EngineRun();

// NETWORK 15
.Engine_Coms();

// NETWORK 16
.Tracking();

// NETWORK 17
.FanCtrl();

// NETWORK 18
.Auto_Sequence();

// NETWORK 19
.ManualSequence();

// NETWORK 20
JackLegs();

// NETWORK 21
Setpoints();

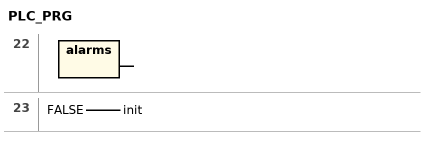
// NETWORK 22
alarms();

// NETWORK 23
init := FALSE;

END_PROGRAM

// StandardPLC/Application/PLC_Version
PROGRAM PLC_Version
VAR
	INIT: BOOL:=TRUE;
	Tx3000: ifmrcan.CAN_Tx;	
	Tx3000_Ton: TON;
	Tx3000_Buffer: ARRAY[0..7] OF USINT := [1,0,3,0,0,0,0,0];	// 1.0.3.0
	Version: SLL_IFM_Version.PLC_Version;	
END_VAR

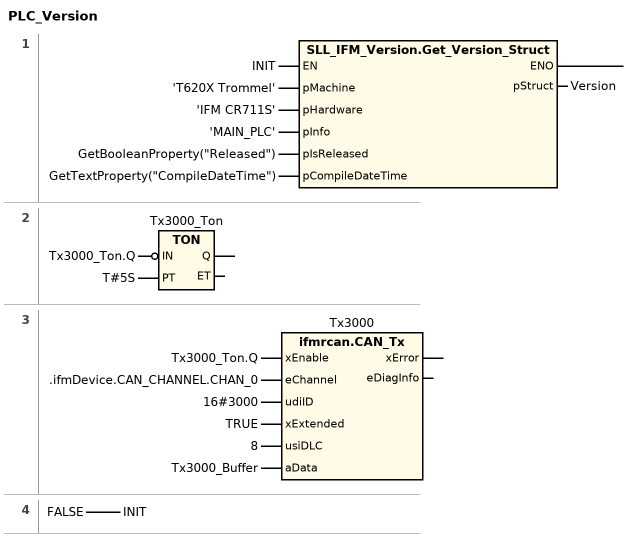
// NETWORK 1
IF INIT THEN
    SLL_IFM_Version.Get_Version_Struct(pMachine := 'T620X Trommel', pHardware := 'IFM CR711S', pInfo := 'MAIN_PLC', pIsReleased := GetBooleanProperty("Released"), pCompileDateTime := GetTextProperty("CompileDateTime"), pStruct => Version);
END_IF

// NETWORK 2
Tx3000_Ton(IN := NOT Tx3000_Ton.Q, PT := T#5S); // TON

// NETWORK 3
Tx3000(
    xEnable := Tx3000_Ton.Q,
    eChannel := .ifmDevice.CAN_CHANNEL.CHAN_0,
    udiID := 16#3000,
    xExtended := TRUE,
    usiDLC := 8,
    aData := Tx3000_Buffer); // ifmrcan.CAN_Tx

// NETWORK 4
INIT := FALSE;

END_PROGRAM

// Project Information/GetBooleanProperty
// This function has been automatically generated from the project information.
{attribute 'signature_flag' := '1073741824'}
{attribute 'register_in_runtime'}
FUNCTION GetBooleanProperty : BOOL
VAR_INPUT
	stKey: WSTRING;
END_VAR

IF stKey = "Released" THEN
	GetBooleanProperty := FALSE;
ELSE
	GetBooleanProperty := FALSE;
END_IF

END_FUNCTION

// Project Information/GetTextProperty
// This function has been automatically generated from the project information.
{attribute 'signature_flag' := '1073741824'}
{attribute 'register_in_runtime'}
FUNCTION GetTextProperty : WSTRING
VAR_INPUT
	stKey: WSTRING;
END_VAR

IF stKey = "Company" THEN
	GetTextProperty := "Mtech";
ELSIF stKey = "Description" THEN
	GetTextProperty := "T620X PLC - pwm ramp mods / sim mods - link fixed for RAMP_LIMIT to the output block";
ELSIF stKey = "Project" THEN
	GetTextProperty := "T620X_PLC_CR711S";
ELSIF stKey = "Title" THEN
	GetTextProperty := "T620X PLC";
ELSE
	GetTextProperty := "";
END_IF

END_FUNCTION

// StandardPLC/Application/SIM_MAIN
PROGRAM SIM_MAIN
VAR
END_VAR

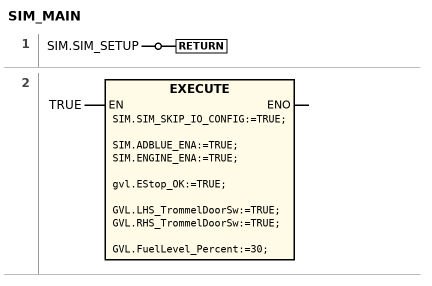
// NETWORK 1
IF NOT SIM.SIM_SETUP THEN RETURN; END_IF

// NETWORK 2
SIM.SIM_SKIP_IO_CONFIG:=TRUE;

SIM.ADBLUE_ENA:=TRUE;
SIM.ENGINE_ENA:=TRUE;

gvl.EStop_OK:=TRUE;

GVL.LHS_TrommelDoorSw:=TRUE;
GVL.RHS_TrommelDoorSw:=TRUE;

GVL.FuelLevel_Percent:=30;

END_PROGRAM

// StandardPLC/Application/config_IO
PROGRAM config_IO
VAR
	IN0100_Input: ifmIOcommon.Input;
	IN0101_Input: ifmIOcommon.Input;
	IN0102_Input: ifmIOcommon.Input;
	IN0103_Input: ifmIOcommon.Input;
	IN0200_Input: ifmIOcommon.Input;
	IN0201_Input: ifmIOcommon.Input;
	IN0202_Input: ifmIOcommon.Input;
	IN0203_Input: ifmIOcommon.Input;
	IN0600_Input: ifmIOcommon.Input;
	IN0601_Input: ifmIOcommon.Input;
	IN0602_Input: ifmIOcommon.Input;
	IN0603_Input: ifmIOcommon.Input;
	IN0700_Input: ifmIOcommon.Input;
	IN0701_Input: ifmIOcommon.Input;
	IN0702_Input: ifmIOcommon.Input;
	IN0703_Input: ifmIOcommon.Input;
	IN0000_Input: ifmIOcommon.Input;
	IN0001_Input: ifmIOcommon.Input;
	IN0002_Input: ifmIOcommon.Input;
	IN0003_Input: ifmIOcommon.Input;
	IN0500_Input: ifmIOcommon.Input;
	IN0501_Input: ifmIOcommon.Input;
	IN0502_Input: ifmIOcommon.Input;
	IN0503_Input: ifmIOcommon.Input;
	IN0400_Input: ifmIOcommon.Input;
	IN0401_Input: ifmIOcommon.Input;
	IN0900_Input: ifmIOcommon.Input;
	IN0901_Input: ifmIOcommon.Input;
	IN0300_Input: ifmIOcommon.Input;
	IN0301_Input: ifmIOcommon.Input;
	IN0800_Input: ifmIOcommon.Input;
	IN0801_Input: ifmIOcommon.Input;
	
	OUT0000_Output: ifmOutPWM.CurrentControl;
	OUT0001_Output: ifmIOcommon.Output;
	OUT0002_Output: ifmOutPWM.CurrentControl;
	OUT0003_Output: ifmIOcommon.Output;
	OUT0004_Output: ifmOutPWM.CurrentControl;
	OUT0005_Output: ifmIOcommon.Output;
	OUT0006_Output: ifmIOcommon.Output;
	OUT0007_Output: ifmOutPWM.CurrentControl;
	OUT0008_Output: ifmIOcommon.Output;
	OUT0100_Output: ifmOutPWM.CurrentControl;
	OUT0101_Output: ifmIOcommon.Output;
	OUT0102_Output: ifmOutPWM.CurrentControl;
	OUT0103_Output: ifmIOcommon.Output;
	OUT0104_Output: ifmIOcommon.Output;
	OUT0105_Output: ifmIOcommon.Output;
	OUT0106_Output: ifmIOcommon.Output;
	OUT0107_Output: ifmIOcommon.Output;
	OUT0108_Output: ifmIOcommon.Output;
	OUT0200_Output: ifmIOcommon.Output;
	OUT0201_Output: ifmIOcommon.Output;
	OUT0202_Output: ifmIOcommon.Output;
	OUT0203_Output: ifmIOcommon.Output;
	OUT0204_Output: ifmIOcommon.Output;
	OUT0205_Output: ifmIOcommon.Output;
	OUT0206_Output: ifmIOcommon.Output;
	OUT0207_Output: ifmIOcommon.Output;
	OUT0208_Output: ifmIOcommon.Output;
	IN401_ScaleBlock: pil.ScaleBlock;
	fbSmoothing_0: fbSmoothing;
	Scale_IN0101: pil.ScaleBlock;
	DrumPressSmooth: fbSmoothing;
	OutputGroup0: ifmOutGroup.OutputGroup;
	OutputGroup1: ifmOutGroup.OutputGroup;
	OutputGroup2: ifmOutGroup.OutputGroup;
END_VAR

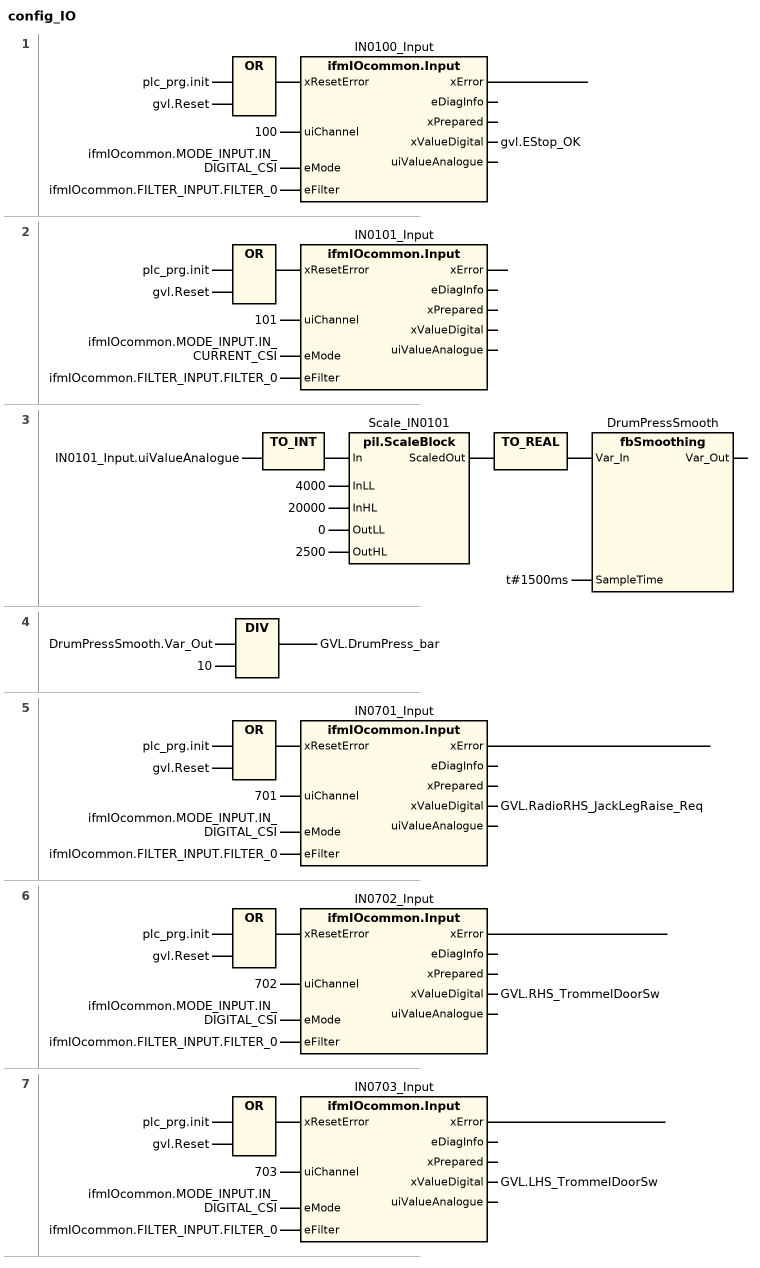
// NETWORK 1
IN0100_Input(
    xResetError := plc_prg.init OR gvl.Reset,
    uiChannel := 100,
    eMode := ifmIOcommon.MODE_INPUT.IN_DIGITAL_CSI,
    eFilter := ifmIOcommon.FILTER_INPUT.FILTER_0,
    xValueDigital => gvl.EStop_OK); // ifmIOcommon.Input

// NETWORK 2
IN0101_Input(
    xResetError := plc_prg.init OR gvl.Reset,
    uiChannel := 101,
    eMode := ifmIOcommon.MODE_INPUT.IN_CURRENT_CSI,
    eFilter := ifmIOcommon.FILTER_INPUT.FILTER_0); // ifmIOcommon.Input

// NETWORK 3
Scale_IN0101(
    In := TO_INT(IN0101_Input.uiValueAnalogue),
    InLL := 4000,
    InHL := 20000,
    OutLL := 0,
    OutHL := 2500); // pil.ScaleBlock
DrumPressSmooth(Var_In := TO_REAL(Scale_IN0101.ScaledOut), SampleTime := t#1500ms); // fbSmoothing

// NETWORK 4
GVL.DrumPress_bar := DrumPressSmooth.Var_Out / 10;

// NETWORK 5
IN0701_Input(
    xResetError := plc_prg.init OR gvl.Reset,
    uiChannel := 701,
    eMode := ifmIOcommon.MODE_INPUT.IN_DIGITAL_CSI,
    eFilter := ifmIOcommon.FILTER_INPUT.FILTER_0,
    xValueDigital => GVL.RadioRHS_JackLegRaise_Req); // ifmIOcommon.Input

// NETWORK 6
IN0702_Input(
    xResetError := plc_prg.init OR gvl.Reset,
    uiChannel := 702,
    eMode := ifmIOcommon.MODE_INPUT.IN_DIGITAL_CSI,
    eFilter := ifmIOcommon.FILTER_INPUT.FILTER_0,
    xValueDigital => GVL.RHS_TrommelDoorSw); // ifmIOcommon.Input

// NETWORK 7
IN0703_Input(
    xResetError := plc_prg.init OR gvl.Reset,
    uiChannel := 703,
    eMode := ifmIOcommon.MODE_INPUT.IN_DIGITAL_CSI,
    eFilter := ifmIOcommon.FILTER_INPUT.FILTER_0,
    xValueDigital => GVL.LHS_TrommelDoorSw); // ifmIOcommon.Input

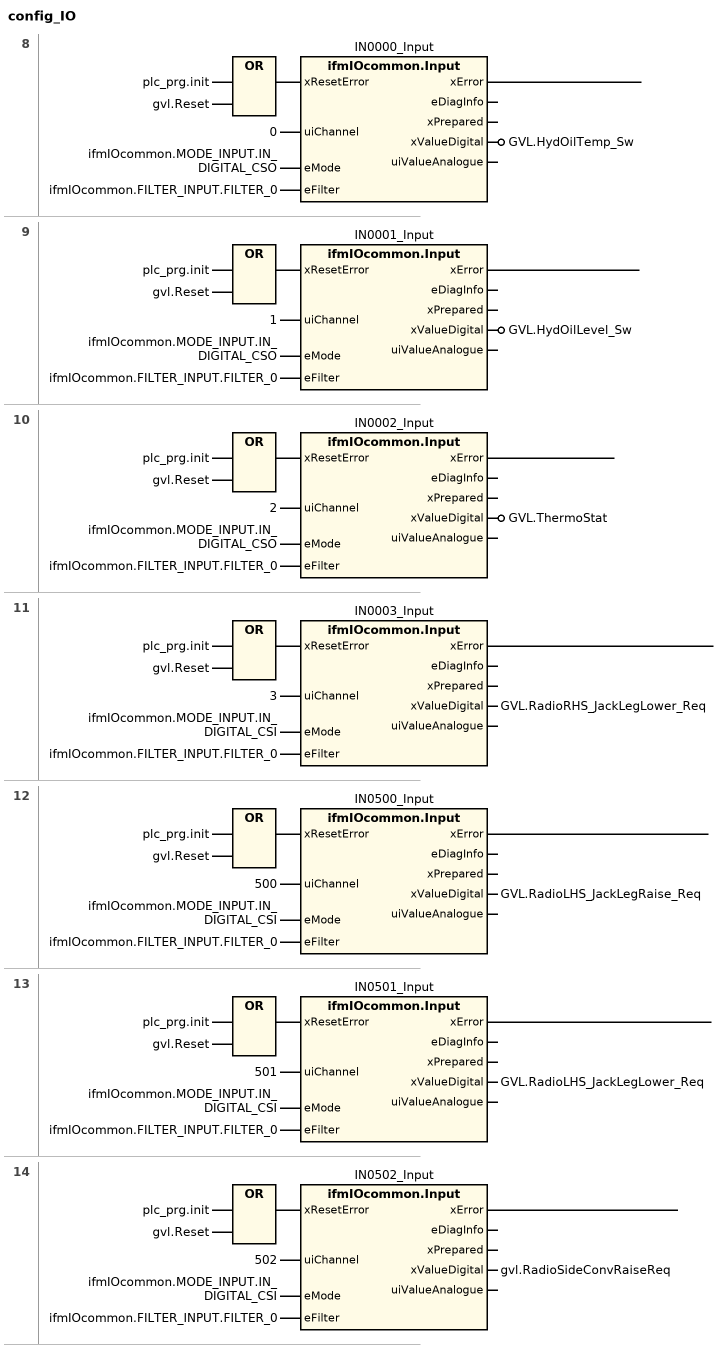
// NETWORK 8
IN0000_Input(
    xResetError := plc_prg.init OR gvl.Reset,
    uiChannel := 0,
    eMode := ifmIOcommon.MODE_INPUT.IN_DIGITAL_CSO,
    eFilter := ifmIOcommon.FILTER_INPUT.FILTER_0); // ifmIOcommon.Input
GVL.HydOilTemp_Sw := NOT IN0000_Input.xValueDigital;

// NETWORK 9
IN0001_Input(
    xResetError := plc_prg.init OR gvl.Reset,
    uiChannel := 1,
    eMode := ifmIOcommon.MODE_INPUT.IN_DIGITAL_CSO,
    eFilter := ifmIOcommon.FILTER_INPUT.FILTER_0); // ifmIOcommon.Input
GVL.HydOilLevel_Sw := NOT IN0001_Input.xValueDigital;

// NETWORK 10
IN0002_Input(
    xResetError := plc_prg.init OR gvl.Reset,
    uiChannel := 2,
    eMode := ifmIOcommon.MODE_INPUT.IN_DIGITAL_CSO,
    eFilter := ifmIOcommon.FILTER_INPUT.FILTER_0); // ifmIOcommon.Input
GVL.ThermoStat := NOT IN0002_Input.xValueDigital;

// NETWORK 11
IN0003_Input(
    xResetError := plc_prg.init OR gvl.Reset,
    uiChannel := 3,
    eMode := ifmIOcommon.MODE_INPUT.IN_DIGITAL_CSI,
    eFilter := ifmIOcommon.FILTER_INPUT.FILTER_0,
    xValueDigital => GVL.RadioRHS_JackLegLower_Req); // ifmIOcommon.Input

// NETWORK 12
IN0500_Input(
    xResetError := plc_prg.init OR gvl.Reset,
    uiChannel := 500,
    eMode := ifmIOcommon.MODE_INPUT.IN_DIGITAL_CSI,
    eFilter := ifmIOcommon.FILTER_INPUT.FILTER_0,
    xValueDigital => GVL.RadioLHS_JackLegRaise_Req); // ifmIOcommon.Input

// NETWORK 13
IN0501_Input(
    xResetError := plc_prg.init OR gvl.Reset,
    uiChannel := 501,
    eMode := ifmIOcommon.MODE_INPUT.IN_DIGITAL_CSI,
    eFilter := ifmIOcommon.FILTER_INPUT.FILTER_0,
    xValueDigital => GVL.RadioLHS_JackLegLower_Req); // ifmIOcommon.Input

// NETWORK 14
IN0502_Input(
    xResetError := plc_prg.init OR gvl.Reset,
    uiChannel := 502,
    eMode := ifmIOcommon.MODE_INPUT.IN_DIGITAL_CSI,
    eFilter := ifmIOcommon.FILTER_INPUT.FILTER_0,
    xValueDigital => gvl.RadioSideConvRaiseReq); // ifmIOcommon.Input

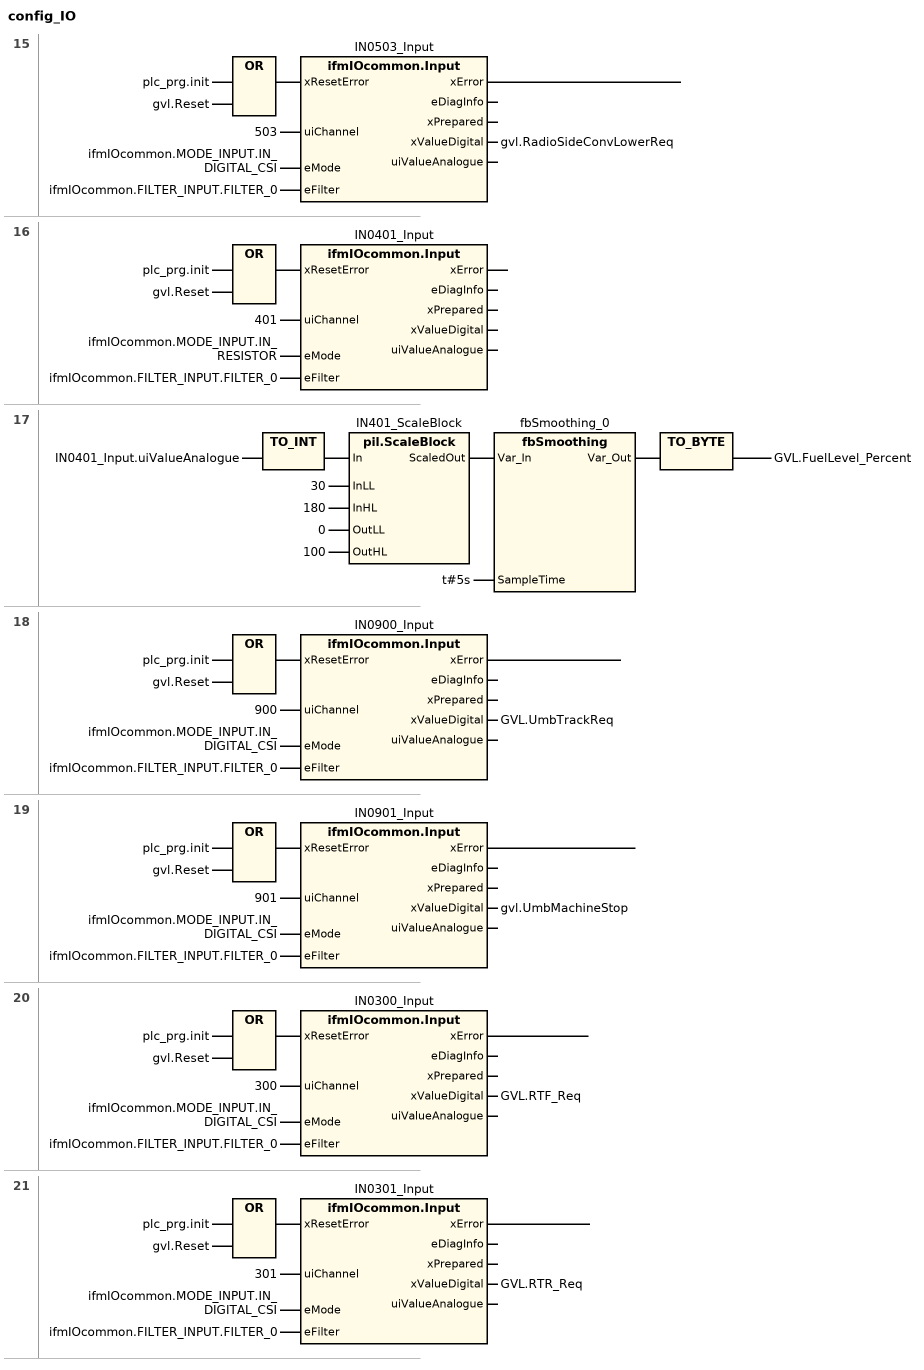
// NETWORK 15
IN0503_Input(
    xResetError := plc_prg.init OR gvl.Reset,
    uiChannel := 503,
    eMode := ifmIOcommon.MODE_INPUT.IN_DIGITAL_CSI,
    eFilter := ifmIOcommon.FILTER_INPUT.FILTER_0,
    xValueDigital => gvl.RadioSideConvLowerReq); // ifmIOcommon.Input

// NETWORK 16
IN0401_Input(
    xResetError := plc_prg.init OR gvl.Reset,
    uiChannel := 401,
    eMode := ifmIOcommon.MODE_INPUT.IN_RESISTOR,
    eFilter := ifmIOcommon.FILTER_INPUT.FILTER_0); // ifmIOcommon.Input

// NETWORK 17
IN401_ScaleBlock(
    In := TO_INT(IN0401_Input.uiValueAnalogue),
    InLL := 30,
    InHL := 180,
    OutLL := 0,
    OutHL := 100); // pil.ScaleBlock
fbSmoothing_0(Var_In := IN401_ScaleBlock.ScaledOut, SampleTime := t#5s); // fbSmoothing
GVL.FuelLevel_Percent := TO_BYTE(fbSmoothing_0.Var_Out);

// NETWORK 18
IN0900_Input(
    xResetError := plc_prg.init OR gvl.Reset,
    uiChannel := 900,
    eMode := ifmIOcommon.MODE_INPUT.IN_DIGITAL_CSI,
    eFilter := ifmIOcommon.FILTER_INPUT.FILTER_0,
    xValueDigital => GVL.UmbTrackReq); // ifmIOcommon.Input

// NETWORK 19
IN0901_Input(
    xResetError := plc_prg.init OR gvl.Reset,
    uiChannel := 901,
    eMode := ifmIOcommon.MODE_INPUT.IN_DIGITAL_CSI,
    eFilter := ifmIOcommon.FILTER_INPUT.FILTER_0,
    xValueDigital => gvl.UmbMachineStop); // ifmIOcommon.Input

// NETWORK 20
IN0300_Input(
    xResetError := plc_prg.init OR gvl.Reset,
    uiChannel := 300,
    eMode := ifmIOcommon.MODE_INPUT.IN_DIGITAL_CSI,
    eFilter := ifmIOcommon.FILTER_INPUT.FILTER_0,
    xValueDigital => GVL.RTF_Req); // ifmIOcommon.Input

// NETWORK 21
IN0301_Input(
    xResetError := plc_prg.init OR gvl.Reset,
    uiChannel := 301,
    eMode := ifmIOcommon.MODE_INPUT.IN_DIGITAL_CSI,
    eFilter := ifmIOcommon.FILTER_INPUT.FILTER_0,
    xValueDigital => GVL.RTR_Req); // ifmIOcommon.Input

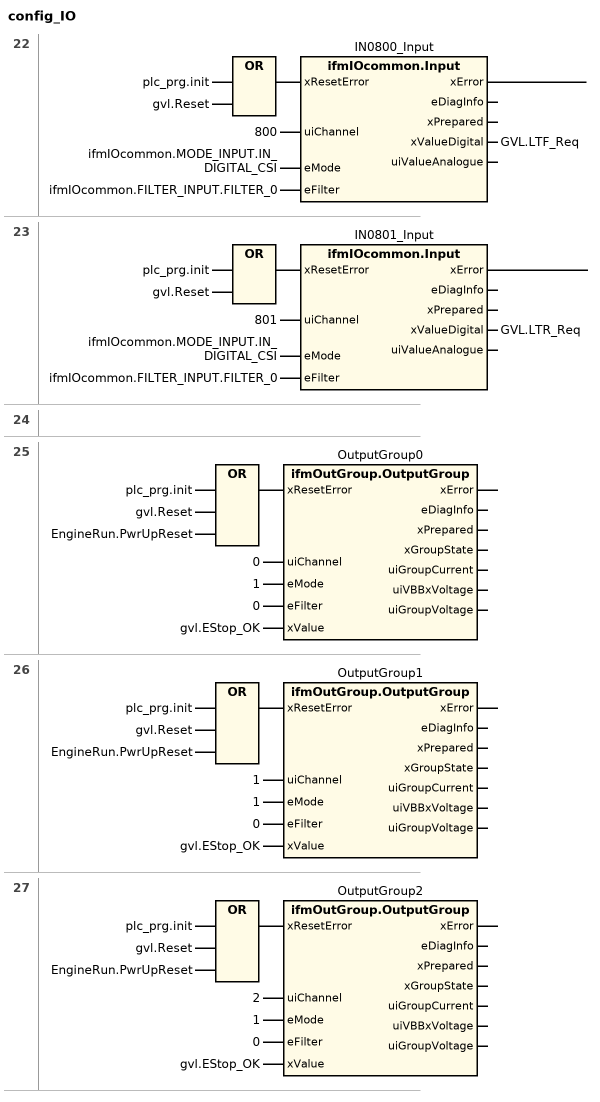
// NETWORK 22
IN0800_Input(
    xResetError := plc_prg.init OR gvl.Reset,
    uiChannel := 800,
    eMode := ifmIOcommon.MODE_INPUT.IN_DIGITAL_CSI,
    eFilter := ifmIOcommon.FILTER_INPUT.FILTER_0,
    xValueDigital => GVL.LTF_Req); // ifmIOcommon.Input

// NETWORK 23
IN0801_Input(
    xResetError := plc_prg.init OR gvl.Reset,
    uiChannel := 801,
    eMode := ifmIOcommon.MODE_INPUT.IN_DIGITAL_CSI,
    eFilter := ifmIOcommon.FILTER_INPUT.FILTER_0,
    xValueDigital => GVL.LTR_Req); // ifmIOcommon.Input

// NETWORK 24

// NETWORK 25
OutputGroup0(
    xResetError := plc_prg.init OR gvl.Reset OR EngineRun.PwrUpReset,
    uiChannel := 0,
    eMode := 1,
    eFilter := 0,
    xValue := gvl.EStop_OK); // ifmOutGroup.OutputGroup

// NETWORK 26
OutputGroup1(
    xResetError := plc_prg.init OR gvl.Reset OR EngineRun.PwrUpReset,
    uiChannel := 1,
    eMode := 1,
    eFilter := 0,
    xValue := gvl.EStop_OK); // ifmOutGroup.OutputGroup

// NETWORK 27
OutputGroup2(
    xResetError := plc_prg.init OR gvl.Reset OR EngineRun.PwrUpReset,
    uiChannel := 2,
    eMode := 1,
    eFilter := 0,
    xValue := gvl.EStop_OK); // ifmOutGroup.OutputGroup

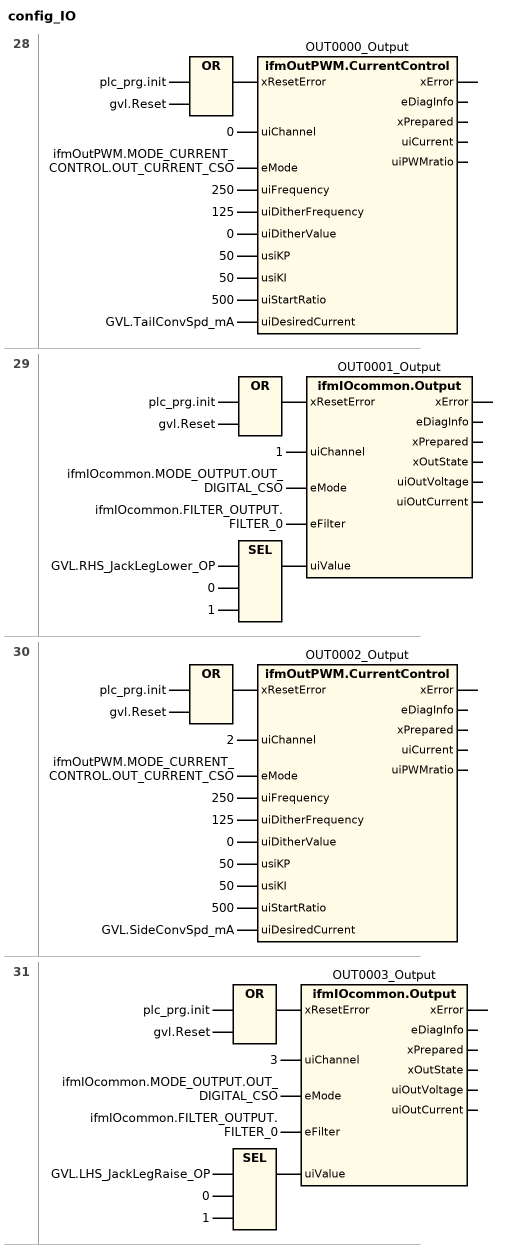
// NETWORK 28
OUT0000_Output(
    xResetError := plc_prg.init OR gvl.Reset,
    uiChannel := 0,
    eMode := ifmOutPWM.MODE_CURRENT_CONTROL.OUT_CURRENT_CSO,
    uiFrequency := 250,
    uiDitherFrequency := 125,
    uiDitherValue := 0,
    usiKP := 50,
    usiKI := 50,
    uiStartRatio := 500,
    uiDesiredCurrent := GVL.TailConvSpd_mA); // ifmOutPWM.CurrentControl

// NETWORK 29
OUT0001_Output(
    xResetError := plc_prg.init OR gvl.Reset,
    uiChannel := 1,
    eMode := ifmIOcommon.MODE_OUTPUT.OUT_DIGITAL_CSO,
    eFilter := ifmIOcommon.FILTER_OUTPUT.FILTER_0,
    uiValue := SEL(GVL.RHS_JackLegLower_OP, 0, 1)); // ifmIOcommon.Output

// NETWORK 30
OUT0002_Output(
    xResetError := plc_prg.init OR gvl.Reset,
    uiChannel := 2,
    eMode := ifmOutPWM.MODE_CURRENT_CONTROL.OUT_CURRENT_CSO,
    uiFrequency := 250,
    uiDitherFrequency := 125,
    uiDitherValue := 0,
    usiKP := 50,
    usiKI := 50,
    uiStartRatio := 500,
    uiDesiredCurrent := GVL.SideConvSpd_mA); // ifmOutPWM.CurrentControl

// NETWORK 31
OUT0003_Output(
    xResetError := plc_prg.init OR gvl.Reset,
    uiChannel := 3,
    eMode := ifmIOcommon.MODE_OUTPUT.OUT_DIGITAL_CSO,
    eFilter := ifmIOcommon.FILTER_OUTPUT.FILTER_0,
    uiValue := SEL(GVL.LHS_JackLegRaise_OP, 0, 1)); // ifmIOcommon.Output

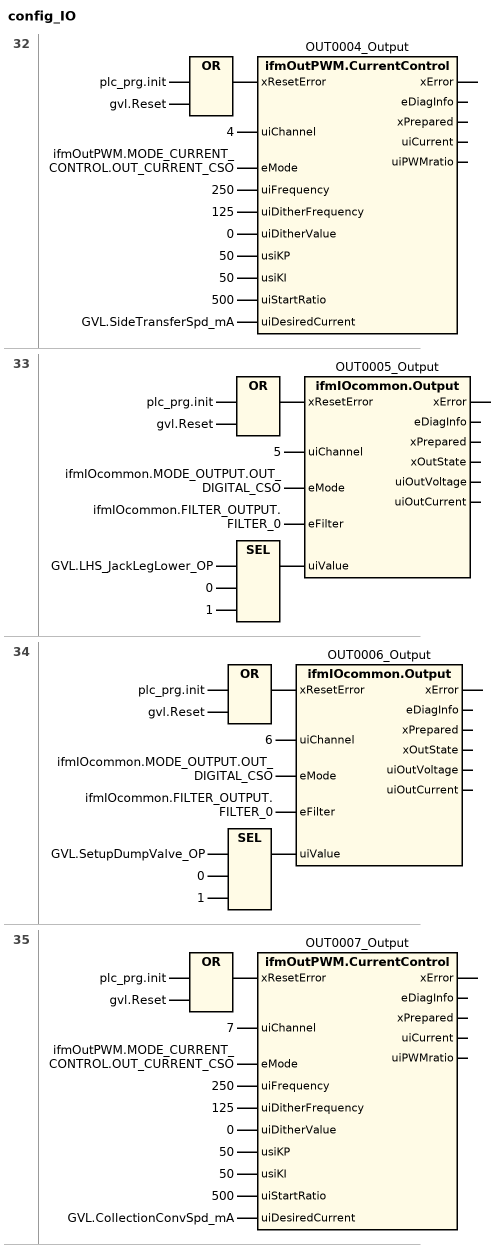
// NETWORK 32
OUT0004_Output(
    xResetError := plc_prg.init OR gvl.Reset,
    uiChannel := 4,
    eMode := ifmOutPWM.MODE_CURRENT_CONTROL.OUT_CURRENT_CSO,
    uiFrequency := 250,
    uiDitherFrequency := 125,
    uiDitherValue := 0,
    usiKP := 50,
    usiKI := 50,
    uiStartRatio := 500,
    uiDesiredCurrent := GVL.SideTransferSpd_mA); // ifmOutPWM.CurrentControl

// NETWORK 33
OUT0005_Output(
    xResetError := plc_prg.init OR gvl.Reset,
    uiChannel := 5,
    eMode := ifmIOcommon.MODE_OUTPUT.OUT_DIGITAL_CSO,
    eFilter := ifmIOcommon.FILTER_OUTPUT.FILTER_0,
    uiValue := SEL(GVL.LHS_JackLegLower_OP, 0, 1)); // ifmIOcommon.Output

// NETWORK 34
OUT0006_Output(
    xResetError := plc_prg.init OR gvl.Reset,
    uiChannel := 6,
    eMode := ifmIOcommon.MODE_OUTPUT.OUT_DIGITAL_CSO,
    eFilter := ifmIOcommon.FILTER_OUTPUT.FILTER_0,
    uiValue := SEL(GVL.SetupDumpValve_OP, 0, 1)); // ifmIOcommon.Output

// NETWORK 35
OUT0007_Output(
    xResetError := plc_prg.init OR gvl.Reset,
    uiChannel := 7,
    eMode := ifmOutPWM.MODE_CURRENT_CONTROL.OUT_CURRENT_CSO,
    uiFrequency := 250,
    uiDitherFrequency := 125,
    uiDitherValue := 0,
    usiKP := 50,
    usiKI := 50,
    uiStartRatio := 500,
    uiDesiredCurrent := GVL.CollectionConvSpd_mA); // ifmOutPWM.CurrentControl

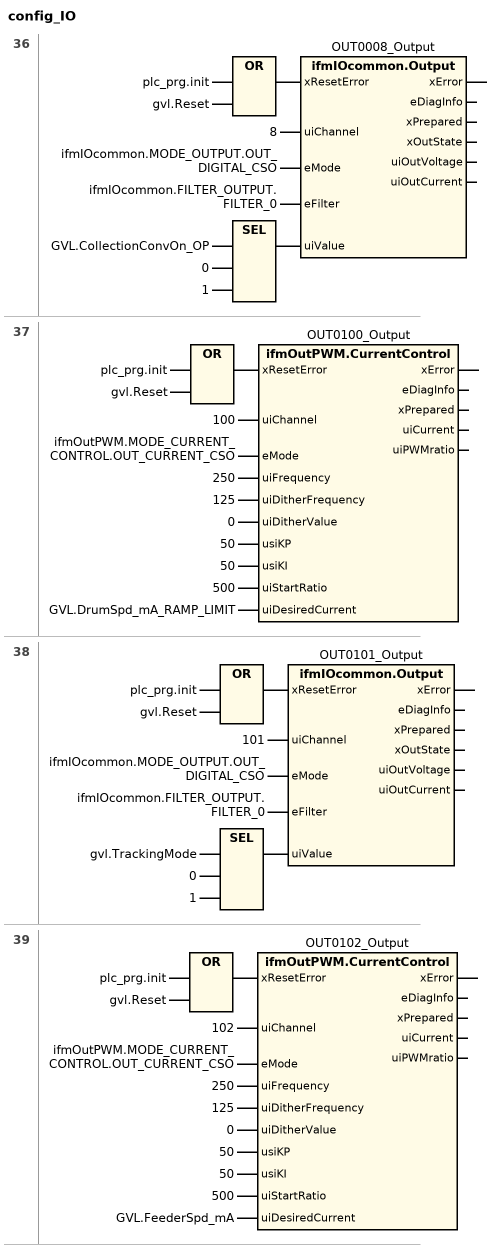
// NETWORK 36
OUT0008_Output(
    xResetError := plc_prg.init OR gvl.Reset,
    uiChannel := 8,
    eMode := ifmIOcommon.MODE_OUTPUT.OUT_DIGITAL_CSO,
    eFilter := ifmIOcommon.FILTER_OUTPUT.FILTER_0,
    uiValue := SEL(GVL.CollectionConvOn_OP, 0, 1)); // ifmIOcommon.Output

// NETWORK 37
OUT0100_Output(
    xResetError := plc_prg.init OR gvl.Reset,
    uiChannel := 100,
    eMode := ifmOutPWM.MODE_CURRENT_CONTROL.OUT_CURRENT_CSO,
    uiFrequency := 250,
    uiDitherFrequency := 125,
    uiDitherValue := 0,
    usiKP := 50,
    usiKI := 50,
    uiStartRatio := 500,
    uiDesiredCurrent := GVL.DrumSpd_mA_RAMP_LIMIT); // ifmOutPWM.CurrentControl

// NETWORK 38
OUT0101_Output(
    xResetError := plc_prg.init OR gvl.Reset,
    uiChannel := 101,
    eMode := ifmIOcommon.MODE_OUTPUT.OUT_DIGITAL_CSO,
    eFilter := ifmIOcommon.FILTER_OUTPUT.FILTER_0,
    uiValue := SEL(gvl.TrackingMode, 0, 1)); // ifmIOcommon.Output

// NETWORK 39
OUT0102_Output(
    xResetError := plc_prg.init OR gvl.Reset,
    uiChannel := 102,
    eMode := ifmOutPWM.MODE_CURRENT_CONTROL.OUT_CURRENT_CSO,
    uiFrequency := 250,
    uiDitherFrequency := 125,
    uiDitherValue := 0,
    usiKP := 50,
    usiKI := 50,
    uiStartRatio := 500,
    uiDesiredCurrent := GVL.FeederSpd_mA); // ifmOutPWM.CurrentControl

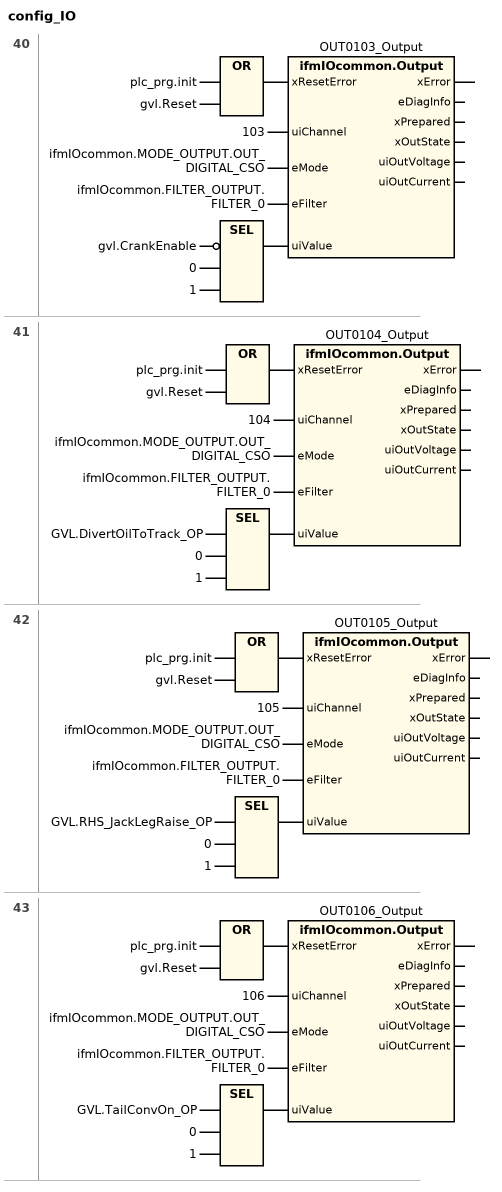
// NETWORK 40
OUT0103_Output(
    xResetError := plc_prg.init OR gvl.Reset,
    uiChannel := 103,
    eMode := ifmIOcommon.MODE_OUTPUT.OUT_DIGITAL_CSO,
    eFilter := ifmIOcommon.FILTER_OUTPUT.FILTER_0,
    uiValue := SEL(NOT gvl.CrankEnable, 0, 1)); // ifmIOcommon.Output

// NETWORK 41
OUT0104_Output(
    xResetError := plc_prg.init OR gvl.Reset,
    uiChannel := 104,
    eMode := ifmIOcommon.MODE_OUTPUT.OUT_DIGITAL_CSO,
    eFilter := ifmIOcommon.FILTER_OUTPUT.FILTER_0,
    uiValue := SEL(GVL.DivertOilToTrack_OP, 0, 1)); // ifmIOcommon.Output

// NETWORK 42
OUT0105_Output(
    xResetError := plc_prg.init OR gvl.Reset,
    uiChannel := 105,
    eMode := ifmIOcommon.MODE_OUTPUT.OUT_DIGITAL_CSO,
    eFilter := ifmIOcommon.FILTER_OUTPUT.FILTER_0,
    uiValue := SEL(GVL.RHS_JackLegRaise_OP, 0, 1)); // ifmIOcommon.Output

// NETWORK 43
OUT0106_Output(
    xResetError := plc_prg.init OR gvl.Reset,
    uiChannel := 106,
    eMode := ifmIOcommon.MODE_OUTPUT.OUT_DIGITAL_CSO,
    eFilter := ifmIOcommon.FILTER_OUTPUT.FILTER_0,
    uiValue := SEL(GVL.TailConvOn_OP, 0, 1)); // ifmIOcommon.Output

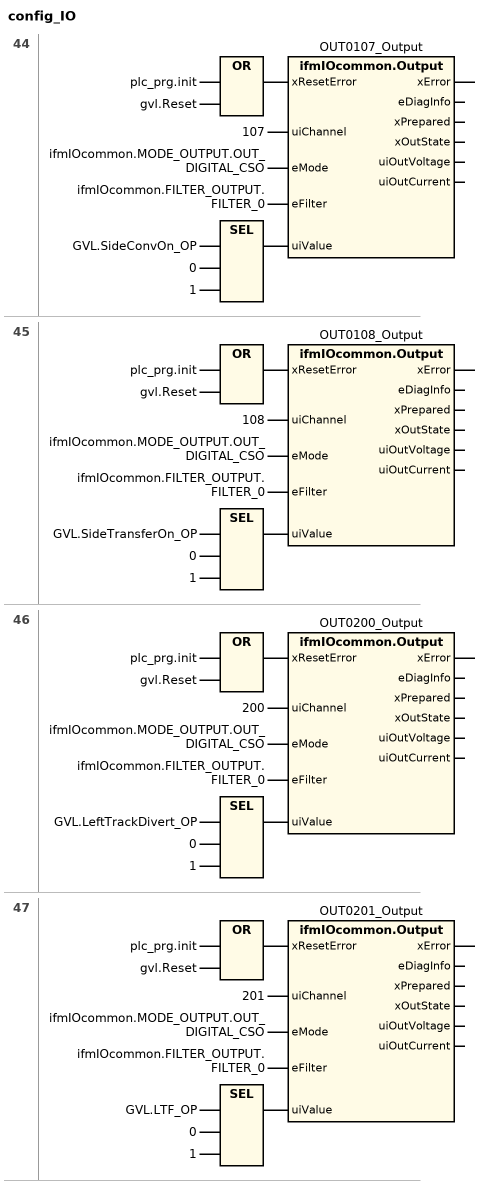
// NETWORK 44
OUT0107_Output(
    xResetError := plc_prg.init OR gvl.Reset,
    uiChannel := 107,
    eMode := ifmIOcommon.MODE_OUTPUT.OUT_DIGITAL_CSO,
    eFilter := ifmIOcommon.FILTER_OUTPUT.FILTER_0,
    uiValue := SEL(GVL.SideConvOn_OP, 0, 1)); // ifmIOcommon.Output

// NETWORK 45
OUT0108_Output(
    xResetError := plc_prg.init OR gvl.Reset,
    uiChannel := 108,
    eMode := ifmIOcommon.MODE_OUTPUT.OUT_DIGITAL_CSO,
    eFilter := ifmIOcommon.FILTER_OUTPUT.FILTER_0,
    uiValue := SEL(GVL.SideTransferOn_OP, 0, 1)); // ifmIOcommon.Output

// NETWORK 46
OUT0200_Output(
    xResetError := plc_prg.init OR gvl.Reset,
    uiChannel := 200,
    eMode := ifmIOcommon.MODE_OUTPUT.OUT_DIGITAL_CSO,
    eFilter := ifmIOcommon.FILTER_OUTPUT.FILTER_0,
    uiValue := SEL(GVL.LeftTrackDivert_OP, 0, 1)); // ifmIOcommon.Output

// NETWORK 47
OUT0201_Output(
    xResetError := plc_prg.init OR gvl.Reset,
    uiChannel := 201,
    eMode := ifmIOcommon.MODE_OUTPUT.OUT_DIGITAL_CSO,
    eFilter := ifmIOcommon.FILTER_OUTPUT.FILTER_0,
    uiValue := SEL(GVL.LTF_OP, 0, 1)); // ifmIOcommon.Output

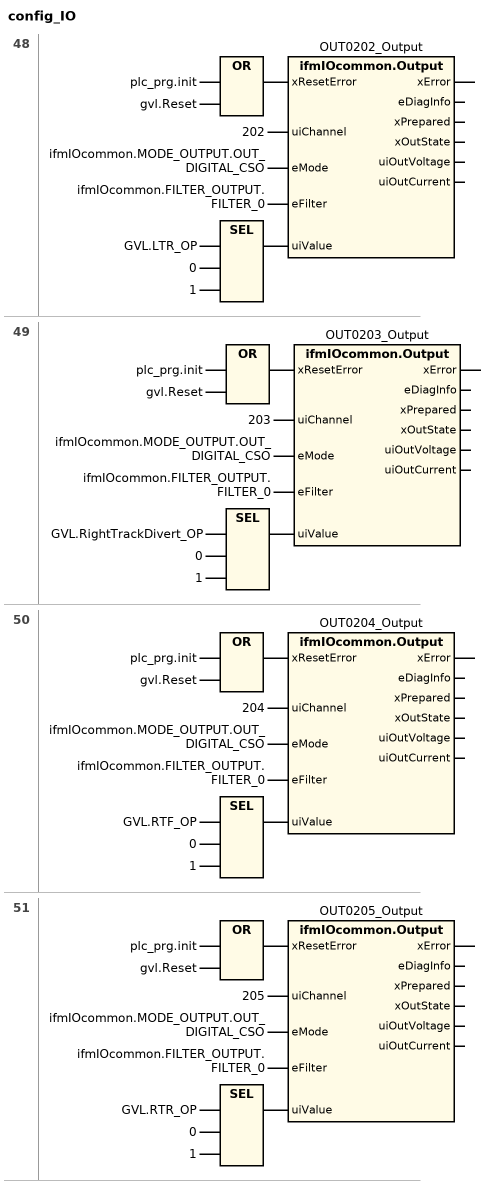
// NETWORK 48
OUT0202_Output(
    xResetError := plc_prg.init OR gvl.Reset,
    uiChannel := 202,
    eMode := ifmIOcommon.MODE_OUTPUT.OUT_DIGITAL_CSO,
    eFilter := ifmIOcommon.FILTER_OUTPUT.FILTER_0,
    uiValue := SEL(GVL.LTR_OP, 0, 1)); // ifmIOcommon.Output

// NETWORK 49
OUT0203_Output(
    xResetError := plc_prg.init OR gvl.Reset,
    uiChannel := 203,
    eMode := ifmIOcommon.MODE_OUTPUT.OUT_DIGITAL_CSO,
    eFilter := ifmIOcommon.FILTER_OUTPUT.FILTER_0,
    uiValue := SEL(GVL.RightTrackDivert_OP, 0, 1)); // ifmIOcommon.Output

// NETWORK 50
OUT0204_Output(
    xResetError := plc_prg.init OR gvl.Reset,
    uiChannel := 204,
    eMode := ifmIOcommon.MODE_OUTPUT.OUT_DIGITAL_CSO,
    eFilter := ifmIOcommon.FILTER_OUTPUT.FILTER_0,
    uiValue := SEL(GVL.RTF_OP, 0, 1)); // ifmIOcommon.Output

// NETWORK 51
OUT0205_Output(
    xResetError := plc_prg.init OR gvl.Reset,
    uiChannel := 205,
    eMode := ifmIOcommon.MODE_OUTPUT.OUT_DIGITAL_CSO,
    eFilter := ifmIOcommon.FILTER_OUTPUT.FILTER_0,
    uiValue := SEL(GVL.RTR_OP, 0, 1)); // ifmIOcommon.Output

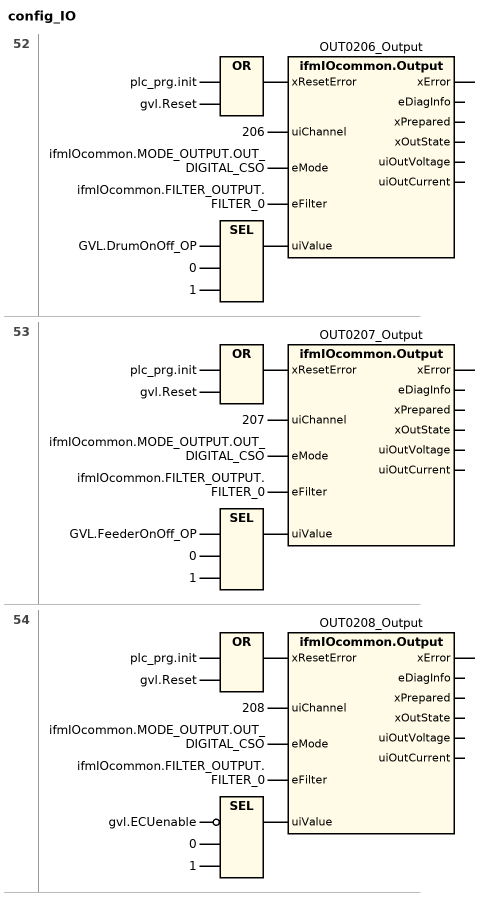
// NETWORK 52
OUT0206_Output(
    xResetError := plc_prg.init OR gvl.Reset,
    uiChannel := 206,
    eMode := ifmIOcommon.MODE_OUTPUT.OUT_DIGITAL_CSO,
    eFilter := ifmIOcommon.FILTER_OUTPUT.FILTER_0,
    uiValue := SEL(GVL.DrumOnOff_OP, 0, 1)); // ifmIOcommon.Output

// NETWORK 53
OUT0207_Output(
    xResetError := plc_prg.init OR gvl.Reset,
    uiChannel := 207,
    eMode := ifmIOcommon.MODE_OUTPUT.OUT_DIGITAL_CSO,
    eFilter := ifmIOcommon.FILTER_OUTPUT.FILTER_0,
    uiValue := SEL(GVL.FeederOnOff_OP, 0, 1)); // ifmIOcommon.Output

// NETWORK 54
OUT0208_Output(
    xResetError := plc_prg.init OR gvl.Reset,
    uiChannel := 208,
    eMode := ifmIOcommon.MODE_OUTPUT.OUT_DIGITAL_CSO,
    eFilter := ifmIOcommon.FILTER_OUTPUT.FILTER_0,
    uiValue := SEL(NOT gvl.ECUenable, 0, 1)); // ifmIOcommon.Output

END_PROGRAM

// StandardPLC/Application/fbSmoothing
FUNCTION_BLOCK fbSmoothing
VAR_INPUT
	Var_In: REAL;
	SampleTime: TIME;
END_VAR
VAR_OUTPUT
	Var_Out: REAL;
END_VAR
VAR
	Timer: TON;
	SampleArray: ARRAY [0..49] OF REAL;
	ArraySampleTime: TIME;
	Timer2: TON;
END_VAR

ArraySampleTime:= SampleTime/50;
Timer(IN:=NOT Timer.Q, PT:=ArraySampleTime, Q=>, ET=> );

IF Timer.Q=TRUE THEN

SampleArray[49]:=SampleArray[48];
SampleArray[48]:=SampleArray[47];
SampleArray[47]:=SampleArray[46];
SampleArray[46]:=SampleArray[45];
SampleArray[45]:=SampleArray[44];
SampleArray[44]:=SampleArray[43];
SampleArray[43]:=SampleArray[42];
SampleArray[42]:=SampleArray[41];
SampleArray[41]:=SampleArray[40];
SampleArray[40]:=SampleArray[39];
SampleArray[39]:=SampleArray[38];
SampleArray[38]:=SampleArray[37];
SampleArray[37]:=SampleArray[36];
SampleArray[36]:=SampleArray[35];
SampleArray[35]:=SampleArray[34];
SampleArray[34]:=SampleArray[33];
SampleArray[33]:=SampleArray[32];
SampleArray[32]:=SampleArray[31];
SampleArray[31]:=SampleArray[30];
SampleArray[30]:=SampleArray[29];
SampleArray[29]:=SampleArray[28];
SampleArray[28]:=SampleArray[27];
SampleArray[27]:=SampleArray[26];
SampleArray[26]:=SampleArray[25];
SampleArray[25]:=SampleArray[24];
SampleArray[24]:=SampleArray[23];
SampleArray[23]:=SampleArray[22];
SampleArray[22]:=SampleArray[21];
SampleArray[21]:=SampleArray[20];
SampleArray[20]:=SampleArray[19];
SampleArray[19]:=SampleArray[18];
SampleArray[18]:=SampleArray[17];
SampleArray[17]:=SampleArray[16];
SampleArray[16]:=SampleArray[15];
SampleArray[15]:=SampleArray[14];
SampleArray[14]:=SampleArray[13];
SampleArray[13]:=SampleArray[12];
SampleArray[12]:=SampleArray[11];
SampleArray[11]:=SampleArray[10];
SampleArray[10]:=SampleArray[9];
SampleArray[9]:=SampleArray[8];
SampleArray[8]:=SampleArray[7];
SampleArray[7]:=SampleArray[6];
SampleArray[6]:=SampleArray[5];
SampleArray[5]:=SampleArray[4];
SampleArray[4]:=SampleArray[3];
SampleArray[3]:=SampleArray[2];
SampleArray[2]:=SampleArray[1];
SampleArray[1]:=SampleArray[0];
SampleArray[0]:=Var_In;
END_IF

Timer2(IN:=NOT Timer2.Q, PT:=SampleTime, Q=>, ET=> );

IF Timer2.Q=TRUE THEN
Var_Out:= (
SampleArray[49] + SampleArray[48] + SampleArray[47] + SampleArray[46] + SampleArray[45] + SampleArray[44] + SampleArray[43] + SampleArray[42] + SampleArray[41] +SampleArray[40] +
SampleArray[39] + SampleArray[38] + SampleArray[37] + SampleArray[36] + SampleArray[35] + SampleArray[34] + SampleArray[33] + SampleArray[32] + SampleArray[31] +SampleArray[30] +
SampleArray[29] + SampleArray[28] + SampleArray[27] + SampleArray[26] + SampleArray[25] + SampleArray[24] + SampleArray[23] + SampleArray[22] + SampleArray[21] +SampleArray[20] +
SampleArray[19] + SampleArray[18] + SampleArray[17] + SampleArray[16] + SampleArray[15] + SampleArray[14] + SampleArray[13] + SampleArray[12] + SampleArray[11] +SampleArray[10] +
SampleArray[9] + SampleArray[8] + SampleArray[7] + SampleArray[6] + SampleArray[5] + SampleArray[4] + SampleArray[3] + SampleArray[2] + SampleArray[1] +SampleArray[0]
			)/50;
END_IF

END_FUNCTION_BLOCK

// StandardPLC/Application/EngineRun
PROGRAM EngineRun
VAR
	TestBit1: BOOL;
	TempWord: WORD;
	TOF_0: tof;
	TestToggle: pil.PB_Toggle;
	PrestartSirenTrig: BOOL;
	PresStartSirenTon: ton;
	PrestartSiren: BOOL;
	FastBlinkWait: ton;
	FastCountBlink: blink;
	FastBlinkTrig: R_trig;
	EngineSpeedPos_Count: SP_CountX1;
	EngineSpeedPos: INT;
	F_TRIG_0: F_Trig;
	R_TRIG_0: R_Trig;
	F_TRIG_1: F_Trig;
	WaitTon1: ton;
	WaitTof1: tof;
	R_TRIG_1: R_Trig;
	TON_0: ton;
	BLINK_0: blink;
	PwrUpReset: BOOL;
END_VAR
VAR // added by the converter: edge detectors and wires of the graphical bodies
    _w1 : BOOL;
END_VAR

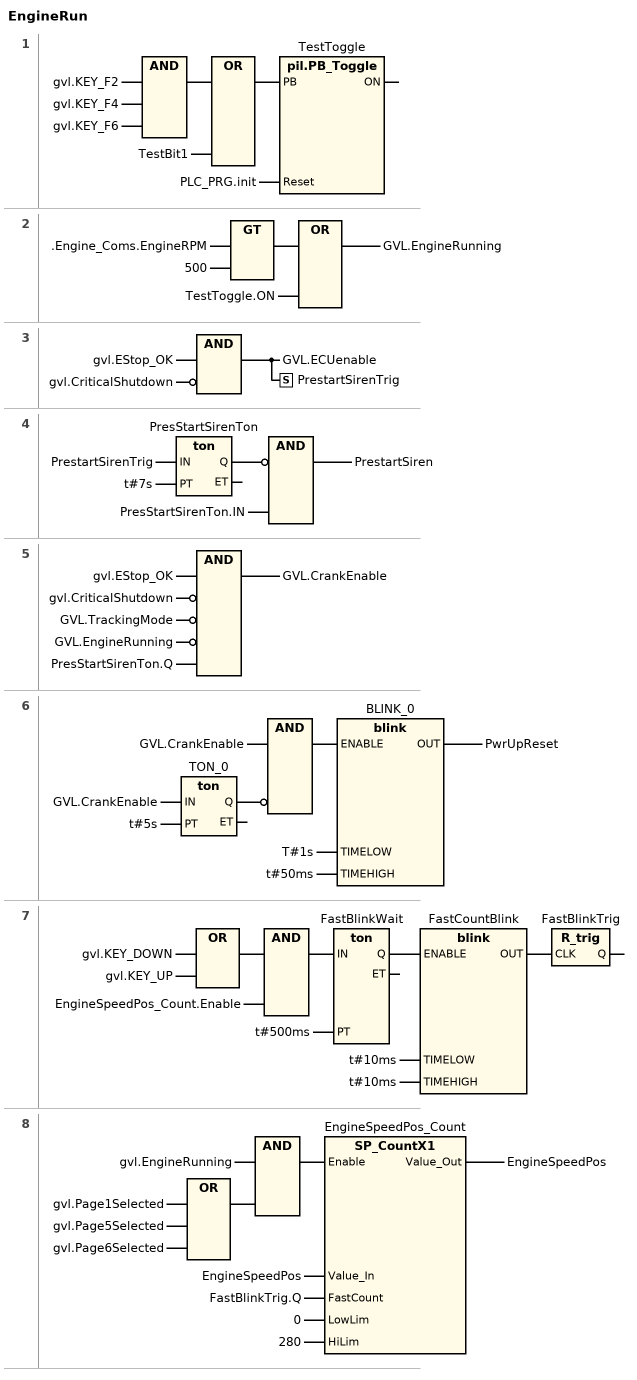
// NETWORK 1
TestToggle(PB := gvl.KEY_F2 AND gvl.KEY_F4 AND gvl.KEY_F6 OR TestBit1, Reset := PLC_PRG.init); // pil.PB_Toggle

// NETWORK 2
GVL.EngineRunning := .Engine_Coms.EngineRPM > 500 OR TestToggle.ON;

// NETWORK 3
_w1 := gvl.EStop_OK AND NOT gvl.CriticalShutdown;
GVL.ECUenable := _w1;
PrestartSirenTrig S= _w1;

// NETWORK 4
PresStartSirenTon(IN := PrestartSirenTrig, PT := t#7s); // ton
PrestartSiren := NOT PresStartSirenTon.Q AND PresStartSirenTon.IN;

// NETWORK 5
GVL.CrankEnable := gvl.EStop_OK AND NOT gvl.CriticalShutdown AND NOT GVL.TrackingMode AND NOT GVL.EngineRunning AND PresStartSirenTon.Q;

// NETWORK 6
TON_0(IN := GVL.CrankEnable, PT := t#5s); // ton
BLINK_0(ENABLE := GVL.CrankEnable AND NOT TON_0.Q, TIMELOW := T#1s, TIMEHIGH := t#50ms); // blink
PwrUpReset := BLINK_0.OUT;

// NETWORK 7
FastBlinkWait(IN := (gvl.KEY_DOWN OR gvl.KEY_UP) AND EngineSpeedPos_Count.Enable, PT := t#500ms); // ton
FastCountBlink(ENABLE := FastBlinkWait.Q, TIMELOW := t#10ms, TIMEHIGH := t#10ms); // blink
FastBlinkTrig(CLK := FastCountBlink.OUT); // R_trig

// NETWORK 8
EngineSpeedPos_Count(
    Enable := gvl.EngineRunning AND (gvl.Page1Selected OR gvl.Page5Selected OR gvl.Page6Selected),
    Value_In := EngineSpeedPos,
    FastCount := FastBlinkTrig.Q,
    LowLim := 0,
    HiLim := 280); // SP_CountX1
EngineSpeedPos := EngineSpeedPos_Count.Value_Out;

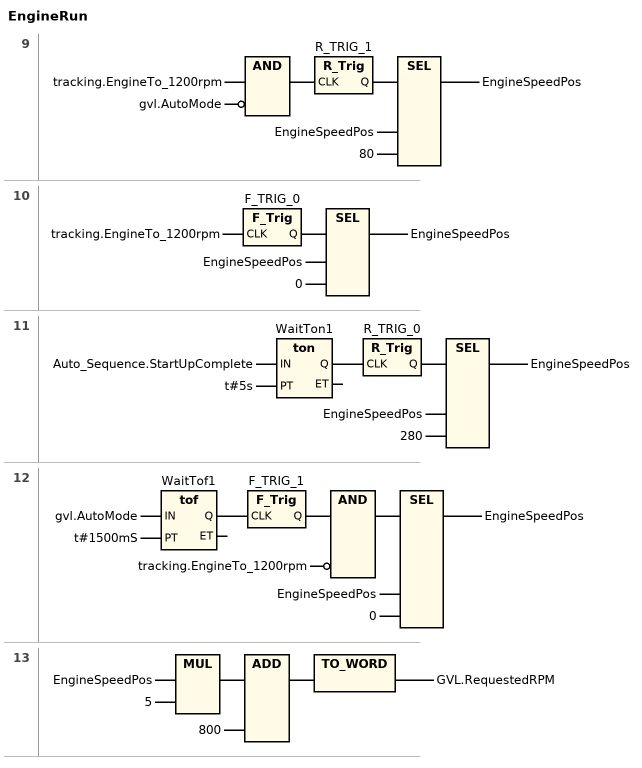
// NETWORK 9
R_TRIG_1(CLK := tracking.EngineTo_1200rpm AND NOT gvl.AutoMode); // R_Trig
EngineSpeedPos := SEL(R_TRIG_1.Q, EngineSpeedPos, 80);

// NETWORK 10
F_TRIG_0(CLK := tracking.EngineTo_1200rpm); // F_Trig
EngineSpeedPos := SEL(F_TRIG_0.Q, EngineSpeedPos, 0);

// NETWORK 11
WaitTon1(IN := Auto_Sequence.StartUpComplete, PT := t#5s); // ton
R_TRIG_0(CLK := WaitTon1.Q); // R_Trig
EngineSpeedPos := SEL(R_TRIG_0.Q, EngineSpeedPos, 280);

// NETWORK 12
WaitTof1(IN := gvl.AutoMode, PT := t#1500mS); // tof
F_TRIG_1(CLK := WaitTof1.Q); // F_Trig
EngineSpeedPos := SEL(F_TRIG_1.Q AND NOT tracking.EngineTo_1200rpm, EngineSpeedPos, 0);

// NETWORK 13
GVL.RequestedRPM := TO_WORD(EngineSpeedPos * 5 + 800);

END_PROGRAM

// StandardPLC/Application/CAN Comms/Engine Comms/Engine_Coms
PROGRAM Engine_Coms
VAR
	EnableCAN1: ifmRCAN.CAN_Enable;
	EngineComsOK: BOOL;
	EngineWarningLamp: BOOL;
	EngineStopLamp: BOOL;
	EngineProtectLamp: BOOL;
	EngineRPM: WORD;
	CoolantTemperature_degC: INT;
	EngineOilPressure_kPa: DWORD;
	CoolantLowLevelWarning: BOOL;
	EngineWaterInFuelWarning: BOOL;
	DM1_Index_Count: CTUD;
	DM1_Index: BYTE;
	DM1_Index_SPN: DWORD;
	DM1_Index_FMI: BYTE;
	DM1_Index_OC: BYTE;
	Flag1: BOOL;
	Tx_TSC1: ifmrcan.CAN_Tx;
	TSC1_Ton1: TON;
	Rx_FECA: ifmrcan.CAN_Rx;
	MILamp: BOOL;
	WtB10: PIL.WordToByte;
	BtDW10: PIL.ByteToDword;
	SPN_Code: DWORD;
	FMI_Code: BYTE;
	OC_Code: BYTE;
	Rx_F004: ifmrcan.CAN_Rx;
	F004_Data: ARRAY [0..7] OF BYTE;
	BtW11: PIL.ByteToWord;
	Rx_FEEE: ifmrcan.CAN_Rx;
	FEEE_Data: ARRAY [0..7] OF BYTE;
	Rx_FEEF: ifmrcan.CAN_Rx;
	FEEF_Data: ARRAY [0..7] OF BYTE;
	FECA_Data: ARRAY [0..7] OF BYTE;
	ECFF_Data: ARRAY [0..7] OF BYTE;
	EBFF_Data: ARRAY [0..7] OF BYTE;
	FF14_Data: ARRAY [0..7] OF BYTE;
	FF0B_Data: ARRAY [0..7] OF BYTE;
	FEE5_Data: ARRAY [0..7] OF BYTE;
	FD7C_Data: ARRAY [0..7] OF BYTE;
	CM: BOOL;
	Rx_ECFF: ifmrcan.CAN_Rx;
	ECFF_RxFlag: BOOL;
	BtDw1: PIL.ByteToDword;
	NumberOfBytes: INT;
	BtW1: PIL.ByteToWord;
	BAM_DM1: BOOL;
	Rx_EBFF: ifmrcan.CAN_Rx;
	EBFF_RxFlag: BOOL;
	LampStatus: BYTE;
	DM1_Array: ARRAY [0..32] OF BYTE;
	EmptyDM1_Array: ARRAY [0..32] OF BYTE :=[ 0,0,0,0,0,0,0,0,0,0,0,0,0,0,0,0,0,0,0,0,0,0,0,0,0,0,0,0,0,0,0,0];
	QtyOf_SPN_Codes: BYTE;
	P2b1: Pack2bits;
	P2b2: Pack2bits;
	P2b3: Pack2bits;
	P2b4: Pack2bits;
	Extract_SPN_1: fb_Extract_SPN;
	Extract_SPN_2: fb_Extract_SPN;
	Extract_SPN_3: fb_Extract_SPN;
	Extract_SPN_4: fb_Extract_SPN;
	Extract_SPN_5: fb_Extract_SPN;
	Extract_SPN_6: fb_Extract_SPN;
	Extract_SPN_7: fb_Extract_SPN;
	Extract_SPN_8: fb_Extract_SPN;
	SPN_Array: ARRAY [1..8] OF DWORD;
	FMI_Array: ARRAY [1..8] OF BYTE;
	OC_Array: ARRAY [1..8] OF BYTE;
	UP1: UNPACK;
	P2b6: Pack2bits;
	P2b7: Pack2bits;
	Tx_Request_PGN: ifmrcan.CAN_Tx;
	RequestWhichPGN_array: ARRAY [0..7] OF BYTE;
	KeyOnWait_1: TON;
	RTrig1: R_TRIG;
	ReqEngHrs_Ton: TON;
	EngHrsReqPulse: BOOL;
	Rx_FEE5: ifmrcan.CAN_Rx;
	BtDw2: PIL.ByteToDword;
	Rx_FD7C: ifmrcan.CAN_Rx;
	DPF_LampStaus: BYTE;
	Tx_CM1: ifmrcan.CAN_Tx;
	RegenInhibit: BOOL;
	CM1_Ton1: TON;
	Standstill_RegenRelease: BOOL;
	RegenInhibit_PBTog: PIL.PB_Toggle;
	ElevateRpmAllowed_PBTog: PIL.PB_Toggle;
	WaitTon2: TON;
	WaitTon3: TON;
	FECA_Rec: BOOL;
	No_Of_Packets: BYTE;
	Packet_Count: CTU;
	TSC1_CheckSum: CounterChecksum;
	Tx_CM2: ifmrcan.CAN_Tx;
	CM2_Ton1: TON;
	DPF_RegenActive: BOOL;
	Coolant_Hi_Temp_DM1: DM1_Condition;
	EngineHiTempWarning: BOOL;
	Oil_Press_Low_DM1: DM1_Condition;
	EngineOilPressWarning: BOOL;
	DPF_Regen_Inhibit1: BOOL;
	P2b8: Pack2bits;
	P2b9: Pack2bits;
	P2b10: Pack2bits;
	DPF_Regen_Inhibit2: BOOL;
	P2b11: Pack2bits;
	DPF_Regen_Inhibit3: BOOL;
	DPF_Regen_Inhibited: BOOL;
	aUSINT_TO_aBYTE_1: PIL.aUSINT_TO_aBYTE;
	aBYTE_TO_aUSINT_0: PIL.aBYTE_TO_aUSINT;
	aUSINT_TO_aBYTE_0: PIL.aUSINT_TO_aBYTE;
	aUSINT_TO_aBYTE_2: PIL.aUSINT_TO_aBYTE;
	aUSINT_TO_aBYTE_3: PIL.aUSINT_TO_aBYTE;
	OilPress_mbar: WORD;
	aUSINT_TO_aBYTE_4: PIL.aUSINT_TO_aBYTE;
	DefTankLevelPercent: BYTE;
	aUSINT_TO_aBYTE_5: PIL.aUSINT_TO_aBYTE;
	EngineHrs: WORD;
	aUSINT_TO_aBYTE_6: PIL.aUSINT_TO_aBYTE;
	aUSINT_TO_aBYTE_7: PIL.aUSINT_TO_aBYTE;
	aUSINT_TO_aBYTE_8: PIL.aUSINT_TO_aBYTE;
	Rx_F003: ifmrcan.CAN_Rx;
	F003_Data: ARRAY [0..7] OF BYTE;

	aUSINT_TO_aBYTE_9: PIL.aUSINT_TO_aBYTE;
	EngineLoadPercent: BYTE;
	Def_Lamp_Status: BYTE;
	DefLowLevLamp: BOOL;
	OilPress_bar: REAL;
	aUSINT_TO_aBYTE_14: PIL.aUSINT_TO_aBYTE;
	Rx_FE56: ifmrcan.CAN_Rx;
	aUSINT_TO_aBYTE_25: PIL.aUSINT_TO_aBYTE;
	FE56_Data: ARRAY [0..7] OF BYTE;

	Rx_FEF2: ifmrcan.CAN_Rx;
	aUSINT_TO_aBYTE_26: PIL.aUSINT_TO_aBYTE;
	FEF2_Data: ARRAY [0..7] OF BYTE;

	BtW12: pil.ByteToWord;
	FuelRate_LHr: REAL;
END_VAR
VAR // added by the converter: edge detectors and wires of the graphical bodies
    _w1, _w2, _w3 : BOOL;
END_VAR

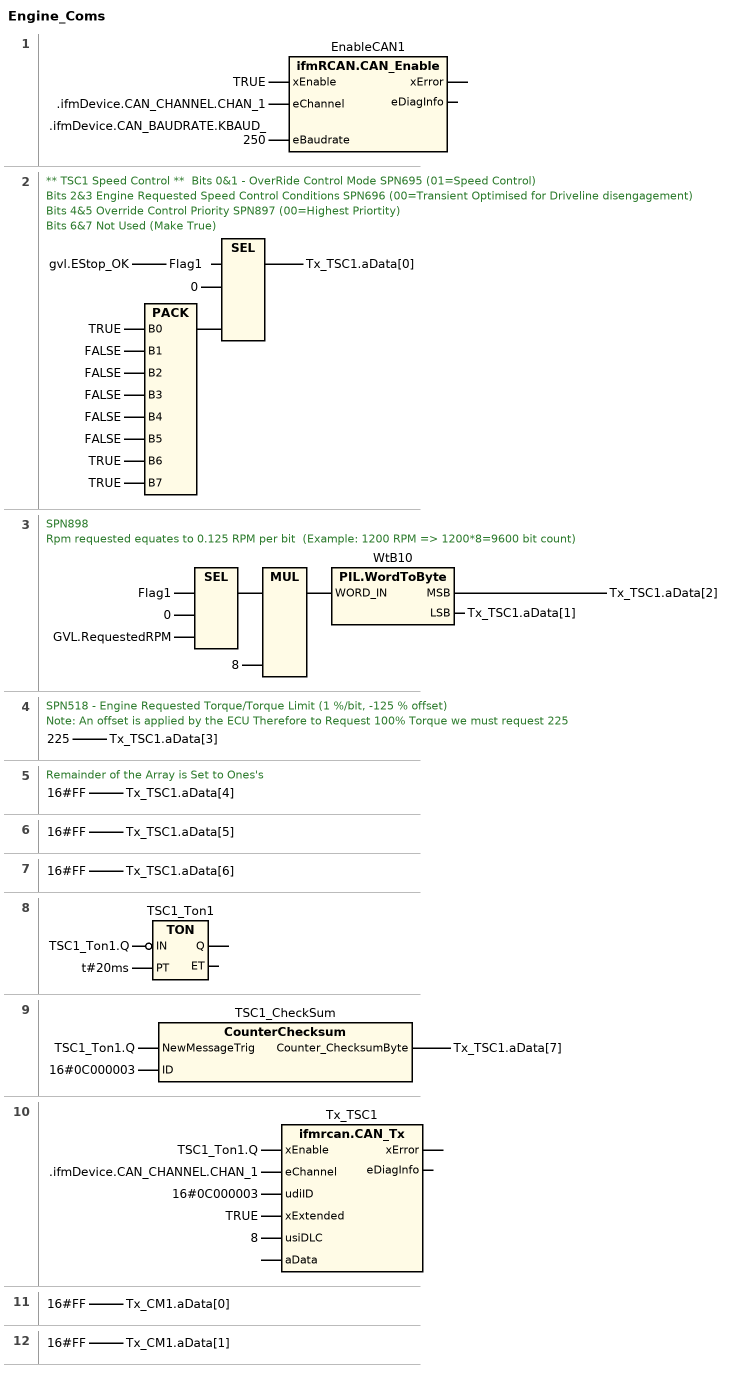
// NETWORK 1
EnableCAN1(
    xEnable := TRUE,
    eChannel := .ifmDevice.CAN_CHANNEL.CHAN_1,
    eBaudrate := .ifmDevice.CAN_BAUDRATE.KBAUD_250); // ifmRCAN.CAN_Enable

// NETWORK 2
// 					** TSC1 Speed Control **  Bits 0&1 - OverRide Control Mode SPN695 (01=Speed Control)
// Bits 2&3 Engine Requested Speed Control Conditions SPN696 (00=Transient Optimised for Driveline disengagement)
// Bits 4&5 Override Control Priority SPN897 (00=Highest Priortity)
// Bits 6&7 Not Used (Make True)
//
Flag1 := gvl.EStop_OK;
Tx_TSC1.aData[0] := SEL(gvl.EStop_OK, 0, PACK(B0 := TRUE, B1 := FALSE, B2 := FALSE, B3 := FALSE, B4 := FALSE, B5 := FALSE, B6 := TRUE, B7 := TRUE));

// NETWORK 3
// 					SPN898
// Rpm requested equates to 0.125 RPM per bit  (Example: 1200 RPM => 1200*8=9600 bit count)
//
WtB10(WORD_IN := SEL(Flag1, 0, GVL.RequestedRPM) * 8, LSB => Tx_TSC1.aData[1]); // PIL.WordToByte
Tx_TSC1.aData[2] := WtB10.MSB;

// NETWORK 4
// 					SPN518 - Engine Requested Torque/Torque Limit (1 %/bit, -125 % offset)
// Note: An offset is applied by the ECU Therefore to Request 100% Torque we must request 225
//
Tx_TSC1.aData[3] := 225;

// NETWORK 5
// Remainder of the Array is Set to Ones's
Tx_TSC1.aData[4] := 16#FF;

// NETWORK 6
Tx_TSC1.aData[5] := 16#FF;

// NETWORK 7
Tx_TSC1.aData[6] := 16#FF;

// NETWORK 8
TSC1_Ton1(IN := NOT TSC1_Ton1.Q, PT := t#20ms); // TON

// NETWORK 9
TSC1_CheckSum(NewMessageTrig := TSC1_Ton1.Q, ID := 16#0C000003); // CounterChecksum
Tx_TSC1.aData[7] := TSC1_CheckSum.Counter_ChecksumByte;

// NETWORK 10
Tx_TSC1(
    xEnable := TSC1_Ton1.Q,
    eChannel := .ifmDevice.CAN_CHANNEL.CHAN_1,
    udiID := 16#0C000003,
    xExtended := TRUE,
    usiDLC := 8); // ifmrcan.CAN_Tx

// NETWORK 11
Tx_CM1.aData[0] := 16#FF;

// NETWORK 12
Tx_CM1.aData[1] := 16#FF;

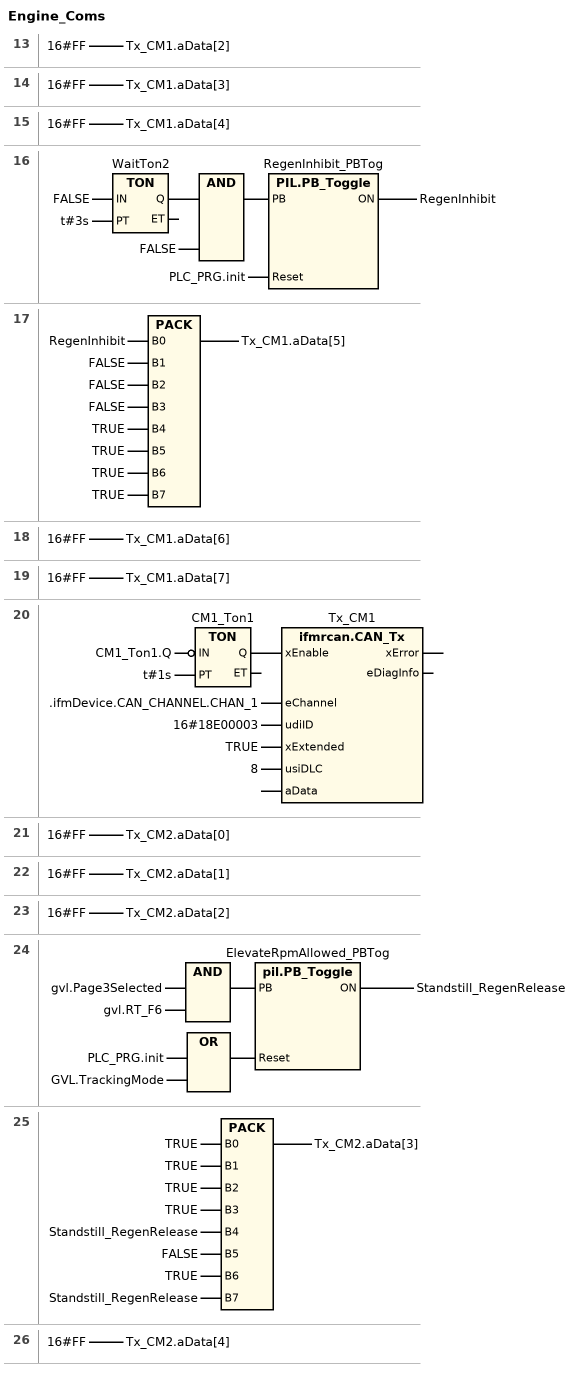
// NETWORK 13
Tx_CM1.aData[2] := 16#FF;

// NETWORK 14
Tx_CM1.aData[3] := 16#FF;

// NETWORK 15
Tx_CM1.aData[4] := 16#FF;

// NETWORK 16
WaitTon2(IN := FALSE, PT := t#3s); // TON
RegenInhibit_PBTog(PB := WaitTon2.Q AND FALSE, Reset := PLC_PRG.init); // PIL.PB_Toggle
RegenInhibit := RegenInhibit_PBTog.ON;

// NETWORK 17
Tx_CM1.aData[5] := PACK(B0 := RegenInhibit, B1 := FALSE, B2 := FALSE, B3 := FALSE, B4 := TRUE, B5 := TRUE, B6 := TRUE, B7 := TRUE);

// NETWORK 18
Tx_CM1.aData[6] := 16#FF;

// NETWORK 19
Tx_CM1.aData[7] := 16#FF;

// NETWORK 20
CM1_Ton1(IN := NOT CM1_Ton1.Q, PT := t#1s); // TON
Tx_CM1(
    xEnable := CM1_Ton1.Q,
    eChannel := .ifmDevice.CAN_CHANNEL.CHAN_1,
    udiID := 16#18E00003,
    xExtended := TRUE,
    usiDLC := 8); // ifmrcan.CAN_Tx

// NETWORK 21
Tx_CM2.aData[0] := 16#FF;

// NETWORK 22
Tx_CM2.aData[1] := 16#FF;

// NETWORK 23
Tx_CM2.aData[2] := 16#FF;

// NETWORK 24
ElevateRpmAllowed_PBTog(PB := gvl.Page3Selected AND gvl.RT_F6, Reset := PLC_PRG.init OR GVL.TrackingMode); // pil.PB_Toggle
Standstill_RegenRelease := ElevateRpmAllowed_PBTog.ON;

// NETWORK 25
Tx_CM2.aData[3] := PACK(B0 := TRUE, B1 := TRUE, B2 := TRUE, B3 := TRUE, B4 := Standstill_RegenRelease, B5 := FALSE, B6 := TRUE, B7 := Standstill_RegenRelease);

// NETWORK 26
Tx_CM2.aData[4] := 16#FF;

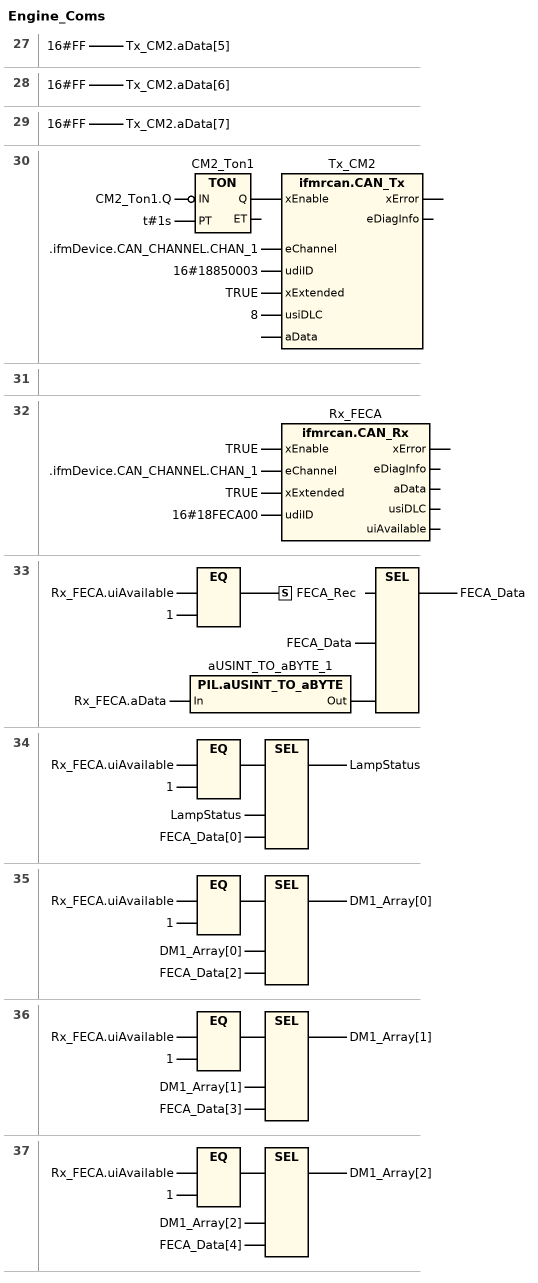
// NETWORK 27
Tx_CM2.aData[5] := 16#FF;

// NETWORK 28
Tx_CM2.aData[6] := 16#FF;

// NETWORK 29
Tx_CM2.aData[7] := 16#FF;

// NETWORK 30
CM2_Ton1(IN := NOT CM2_Ton1.Q, PT := t#1s); // TON
Tx_CM2(
    xEnable := CM2_Ton1.Q,
    eChannel := .ifmDevice.CAN_CHANNEL.CHAN_1,
    udiID := 16#18850003,
    xExtended := TRUE,
    usiDLC := 8); // ifmrcan.CAN_Tx

// NETWORK 31

// NETWORK 32
Rx_FECA(xEnable := TRUE, eChannel := .ifmDevice.CAN_CHANNEL.CHAN_1, xExtended := TRUE, udiID := 16#18FECA00); // ifmrcan.CAN_Rx

// NETWORK 33
_w1 := Rx_FECA.uiAvailable = 1;
FECA_Rec S= _w1;
aUSINT_TO_aBYTE_1(In := Rx_FECA.aData); // PIL.aUSINT_TO_aBYTE
FECA_Data := SEL(_w1, FECA_Data, aUSINT_TO_aBYTE_1.Out);

// NETWORK 34
LampStatus := SEL(Rx_FECA.uiAvailable = 1, LampStatus, FECA_Data[0]);

// NETWORK 35
DM1_Array[0] := SEL(Rx_FECA.uiAvailable = 1, DM1_Array[0], FECA_Data[2]);

// NETWORK 36
DM1_Array[1] := SEL(Rx_FECA.uiAvailable = 1, DM1_Array[1], FECA_Data[3]);

// NETWORK 37
DM1_Array[2] := SEL(Rx_FECA.uiAvailable = 1, DM1_Array[2], FECA_Data[4]);

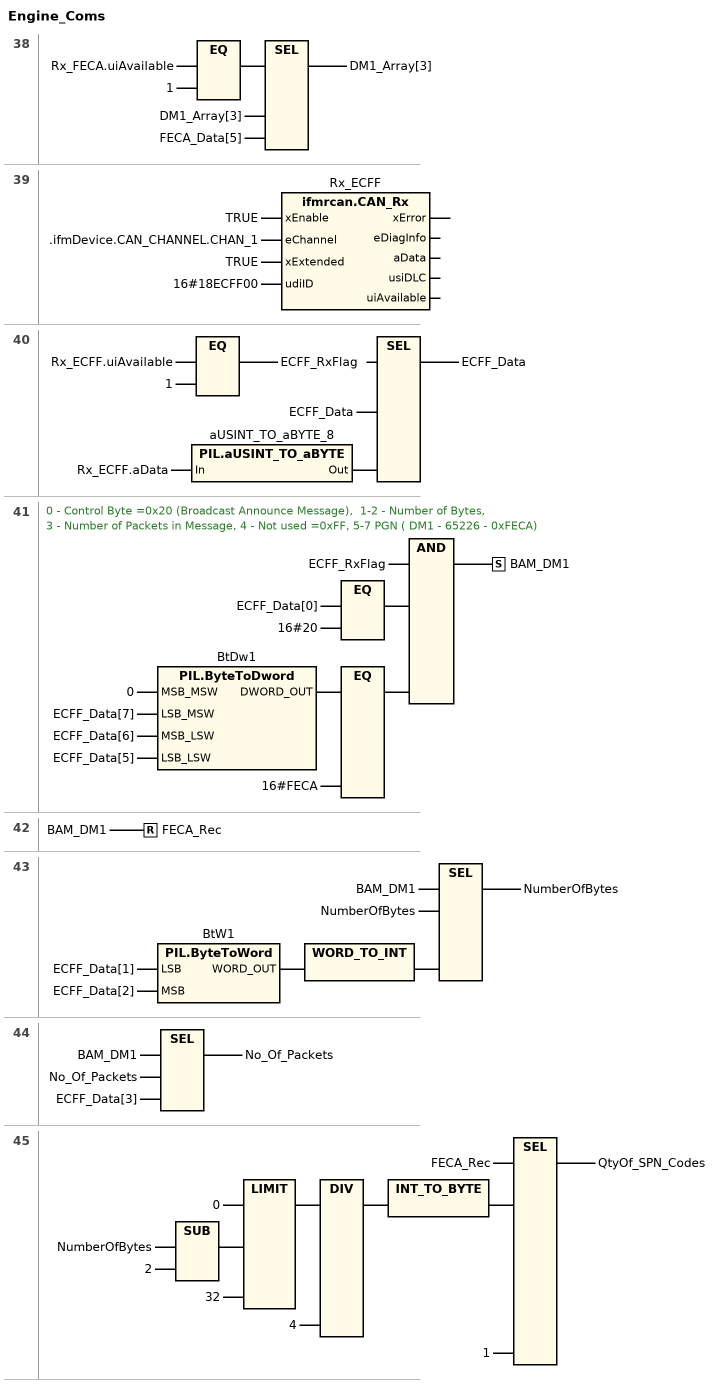
// NETWORK 38
DM1_Array[3] := SEL(Rx_FECA.uiAvailable = 1, DM1_Array[3], FECA_Data[5]);

// NETWORK 39
Rx_ECFF(xEnable := TRUE, eChannel := .ifmDevice.CAN_CHANNEL.CHAN_1, xExtended := TRUE, udiID := 16#18ECFF00); // ifmrcan.CAN_Rx

// NETWORK 40
_w2 := Rx_ECFF.uiAvailable = 1;
ECFF_RxFlag := _w2;
aUSINT_TO_aBYTE_8(In := Rx_ECFF.aData); // PIL.aUSINT_TO_aBYTE
ECFF_Data := SEL(_w2, ECFF_Data, aUSINT_TO_aBYTE_8.Out);

// NETWORK 41
// 					0 - Control Byte =0x20 (Broadcast Announce Message),  1-2 - Number of Bytes,
// 3 - Number of Packets in Message, 4 - Not used =0xFF, 5-7 PGN ( DM1 - 65226 - 0xFECA)
//
BtDw1(MSB_MSW := 0, LSB_MSW := ECFF_Data[7], MSB_LSW := ECFF_Data[6], LSB_LSW := ECFF_Data[5]); // PIL.ByteToDword
BAM_DM1 S= ECFF_RxFlag AND ECFF_Data[0] = 16#20 AND BtDw1.DWORD_OUT = 16#FECA;

// NETWORK 42
FECA_Rec R= BAM_DM1;

// NETWORK 43
BtW1(LSB := ECFF_Data[1], MSB := ECFF_Data[2]); // PIL.ByteToWord
NumberOfBytes := SEL(BAM_DM1, NumberOfBytes, WORD_TO_INT(BtW1.WORD_OUT));

// NETWORK 44
No_Of_Packets := SEL(BAM_DM1, No_Of_Packets, ECFF_Data[3]);

// NETWORK 45
QtyOf_SPN_Codes := SEL(FECA_Rec, INT_TO_BYTE(LIMIT(0, NumberOfBytes - 2, 32) / 4), 1);

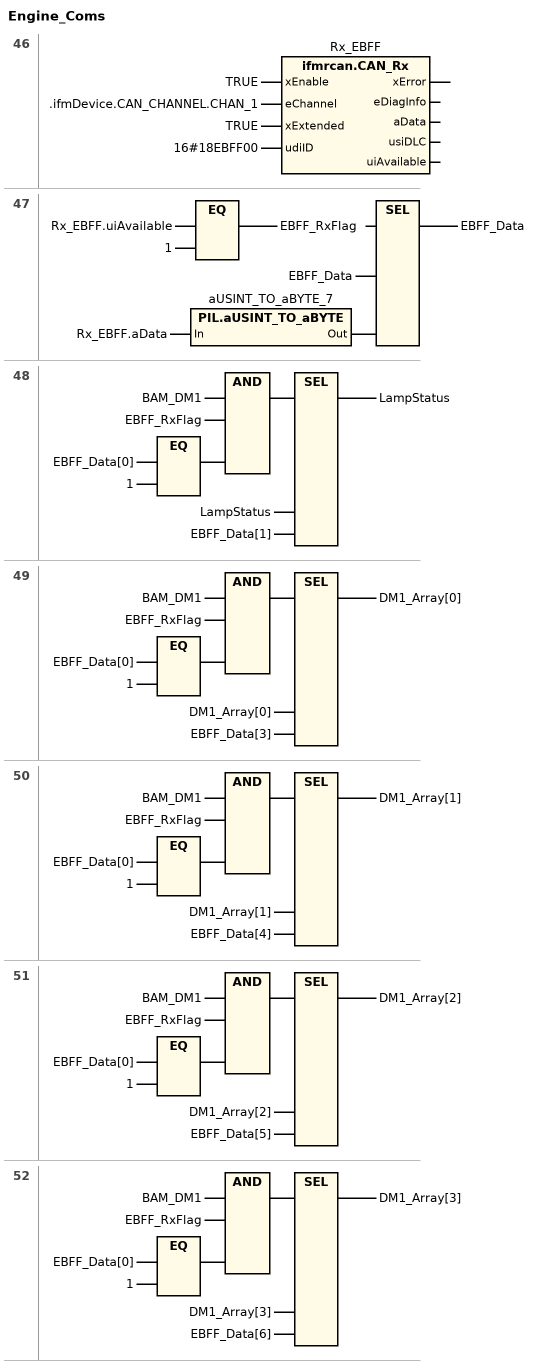
// NETWORK 46
Rx_EBFF(xEnable := TRUE, eChannel := .ifmDevice.CAN_CHANNEL.CHAN_1, xExtended := TRUE, udiID := 16#18EBFF00); // ifmrcan.CAN_Rx

// NETWORK 47
_w3 := Rx_EBFF.uiAvailable = 1;
EBFF_RxFlag := _w3;
aUSINT_TO_aBYTE_7(In := Rx_EBFF.aData); // PIL.aUSINT_TO_aBYTE
EBFF_Data := SEL(_w3, EBFF_Data, aUSINT_TO_aBYTE_7.Out);

// NETWORK 48
LampStatus := SEL(BAM_DM1 AND EBFF_RxFlag AND EBFF_Data[0] = 1, LampStatus, EBFF_Data[1]);

// NETWORK 49
DM1_Array[0] := SEL(BAM_DM1 AND EBFF_RxFlag AND EBFF_Data[0] = 1, DM1_Array[0], EBFF_Data[3]);

// NETWORK 50
DM1_Array[1] := SEL(BAM_DM1 AND EBFF_RxFlag AND EBFF_Data[0] = 1, DM1_Array[1], EBFF_Data[4]);

// NETWORK 51
DM1_Array[2] := SEL(BAM_DM1 AND EBFF_RxFlag AND EBFF_Data[0] = 1, DM1_Array[2], EBFF_Data[5]);

// NETWORK 52
DM1_Array[3] := SEL(BAM_DM1 AND EBFF_RxFlag AND EBFF_Data[0] = 1, DM1_Array[3], EBFF_Data[6]);

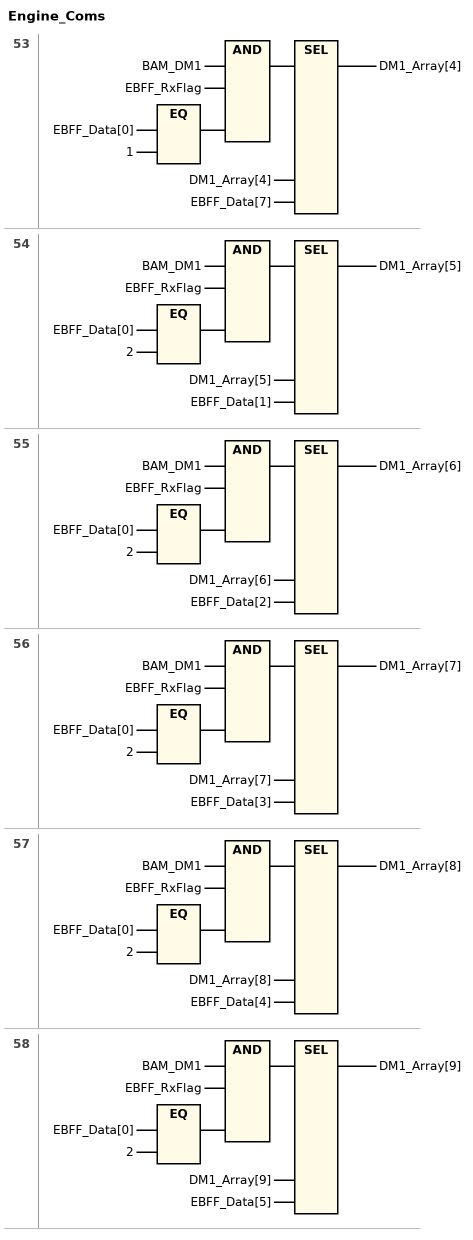
// NETWORK 53
DM1_Array[4] := SEL(BAM_DM1 AND EBFF_RxFlag AND EBFF_Data[0] = 1, DM1_Array[4], EBFF_Data[7]);

// NETWORK 54
DM1_Array[5] := SEL(BAM_DM1 AND EBFF_RxFlag AND EBFF_Data[0] = 2, DM1_Array[5], EBFF_Data[1]);

// NETWORK 55
DM1_Array[6] := SEL(BAM_DM1 AND EBFF_RxFlag AND EBFF_Data[0] = 2, DM1_Array[6], EBFF_Data[2]);

// NETWORK 56
DM1_Array[7] := SEL(BAM_DM1 AND EBFF_RxFlag AND EBFF_Data[0] = 2, DM1_Array[7], EBFF_Data[3]);

// NETWORK 57
DM1_Array[8] := SEL(BAM_DM1 AND EBFF_RxFlag AND EBFF_Data[0] = 2, DM1_Array[8], EBFF_Data[4]);

// NETWORK 58
DM1_Array[9] := SEL(BAM_DM1 AND EBFF_RxFlag AND EBFF_Data[0] = 2, DM1_Array[9], EBFF_Data[5]);

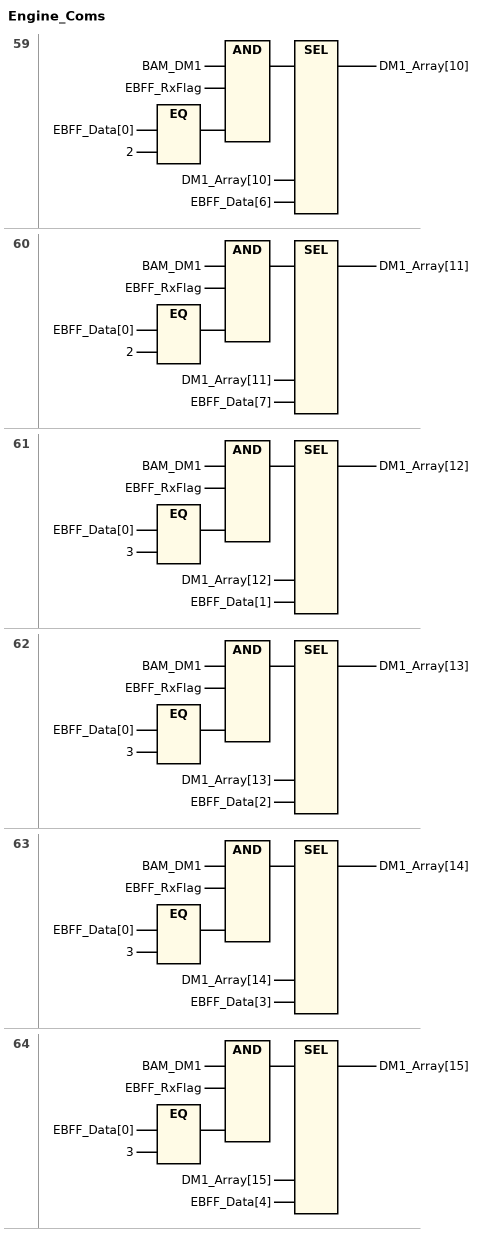
// NETWORK 59
DM1_Array[10] := SEL(BAM_DM1 AND EBFF_RxFlag AND EBFF_Data[0] = 2, DM1_Array[10], EBFF_Data[6]);

// NETWORK 60
DM1_Array[11] := SEL(BAM_DM1 AND EBFF_RxFlag AND EBFF_Data[0] = 2, DM1_Array[11], EBFF_Data[7]);

// NETWORK 61
DM1_Array[12] := SEL(BAM_DM1 AND EBFF_RxFlag AND EBFF_Data[0] = 3, DM1_Array[12], EBFF_Data[1]);

// NETWORK 62
DM1_Array[13] := SEL(BAM_DM1 AND EBFF_RxFlag AND EBFF_Data[0] = 3, DM1_Array[13], EBFF_Data[2]);

// NETWORK 63
DM1_Array[14] := SEL(BAM_DM1 AND EBFF_RxFlag AND EBFF_Data[0] = 3, DM1_Array[14], EBFF_Data[3]);

// NETWORK 64
DM1_Array[15] := SEL(BAM_DM1 AND EBFF_RxFlag AND EBFF_Data[0] = 3, DM1_Array[15], EBFF_Data[4]);

